THIS^.testisEqualToIgnoreCase(
	stringToTest := 'UPPERCASE',
	expectedString := 'UPPERCASE'
);
THIS^.testisEqualToIgnoreCase(
	stringToTest := 'lowercase',
	expectedString := 'lowercase'
);
THIS^.testisEqualToIgnoreCase(
	stringToTest := 'UPPERCASE',
	expectedString := 'lowercase'
);
THIS^.testisEqualToIgnoreCase(
	stringToTest := 'lowercase',
	expectedString := 'UPPERCASE'
);
THIS^.testisEqualToIgnoreCase(
	stringToTest := 'lowercase$80$B9$C6$D4',
	expectedString := 'CASE$80$B9$C6$D4'
);

TcUnit.TEST_FINISHED();
END_METHOD

(*
short summary
==================
This test method tests ``assert.string.windows125x.IsNotEmpty``
method of CNM_AssertionInterfaces library with various inputs

.. <legal notes>

legal notes
=================
| SPDX-FileCopyrightText: © 2022 ekvip automation GmbH <info@ekvip.de>
| SPDX-License-Identifier: Apache-2.0
| For details check: Apache-2.0_

.. _Apache-2.0: https://www.apache.org/licenses/LICENSE-2.0

.. </legal notes>

*)

METHOD runIsNotEmpty : BOOL
VAR_INPUT
END_VAR
RETURN (NOT TcUnit.TEST_ORDERED(THIS^.getTestNameFor('IsNotEmpty')));

THIS^.testIsNotEmpty(
	stringToTest := ''
);
THIS^.testIsNotEmpty(
	stringToTest := 'not empty'
);
THIS^.testIsNotEmpty(
	stringToTest := '{|}~'
);
THIS^.testIsNotEmpty(
	stringToTest := '3649213469328'
);
THIS^.testIsNotEmpty(
	stringToTest := '1one!'
);
THIS^.testIsNotEmpty(
	stringToTest := '$40$n$t$$$"$''
);
THIS^.testIsNotEmpty(
	stringToTest := '$n$t'
);
THIS^.testIsEmpty(
	stringToTest := '$80$8C$A9$B9$C6$D4$F4$7E',
);
THIS^.testIsNotEmpty(
	stringToTest := 'frontmiddleback'
);
THIS^.testIsNotEmpty(
	stringToTest := 'backfrontmiddle'
);
THIS^.testIsNotEmpty(
	stringToTest := 'J;%_iTxQSk?6GfWewt}yMKh1)VXqPA@P1YQ:{EAg:8VJ,/FM;j)xJ[[AvYp/}}SzEgtfYS,1K0.5VtA+VJrB(p#55h2z##mw#F)Y@P6Jz9G@6vb=x#E!cYk(Svr@S*KiPJr1VZ6AjrNback4G=vBJd.E:=,k3!wmuGDe#ZKMD#Vx%?M_0&L0#vT]J,+)ZvU{w%8X0=:XzthmT0VG0QrwpXXCWpFxu6[b!c.BunYYfLQi.,?ut?-{jrC1phTHL)y'
);

TcUnit.TEST_FINISHED();
END_METHOD

(*
short summary
==================
This test method tests ``assert.string.windows125x.isNotEqualTo``
method of CNM_AssertionInterfaces library with various inputs

.. <legal notes>

legal notes
=================
| SPDX-FileCopyrightText: © 2022 ekvip automation GmbH <info@ekvip.de>
| SPDX-License-Identifier: Apache-2.0
| For details check: Apache-2.0_

.. _Apache-2.0: https://www.apache.org/licenses/LICENSE-2.0

.. </legal notes>

*)


METHOD runIsNotEqualTo : BOOL
VAR_INPUT
END_VAR
RETURN (NOT TcUnit.TEST_ORDERED(THIS^.getTestNameFor('isNotEqualTo')));

THIS^.testisNotEqualTo(
	stringToTest := '',
	expectedString := ''
);
THIS^.testisNotEqualTo(
	stringToTest := 'not empty',
	expectedString := ''
);
THIS^.testisNotEqualTo(
	stringToTest := '',
	expectedString := 'not empty'
);
THIS^.testisNotEqualTo(
	stringToTest := 'not empty',
	expectedString := 'not'
);
THIS^.testisNotEqualTo(
	stringToTest := 'not empty',
	expectedString := 'not empty'
);
THIS^.testisNotEqualTo(
	stringToTest := '{|}~',
	expectedString := '3649213469328'
);
THIS^.testisNotEqualTo(
	stringToTest := '1one!',
	expectedString := '1one'
);
THIS^.testisNotEqualTo(
	stringToTest := '1one!',
	expectedString := '1one!'
);

THIS^.testisNotEqualTo(
	stringToTest := '$40$n$t$$$"$'',
	expectedString := '$n$t'
);
THIS^.testisNotEqualTo(
	stringToTest := '$40$n$t$$$"$'',
	expectedString := '$40$n$t$$$"$''
);
THIS^.testIsNotEqualTo(
	stringToTest := '$80$8C$A9$B9$C6$D4$F4$7E',
	expectedString := '$B9$C6$D4'
);
THIS^.testIsNotEqualTo(
	stringToTest := '$80$8C$A9$B9$C6$D4$F4$7E',
	expectedString := '$80$B9$C6$D4'
);
THIS^.testisNotEqualTo(
	stringToTest := 'frontmiddleback',
	expectedString := 'back'
);
THIS^.testisNotEqualTo(
	stringToTest := 'frontmiddleback',
	expectedString := 'frontmiddlebackfront'
);
THIS^.testisNotEqualTo(
	stringToTest := 'backfrontmiddle',
	expectedString := 'backmiddle'
);
THIS^.testisNotEqualTo(
	stringToTest := 'J;%_iTxQSk?6GfWewt}yMKh1)VXqPA@P1YQ:{EAg:8VJ,/FM;j)xJ[[AvYp/}}SzEgtfYS,1K0.5VtA+VJrB(p#55h2z##mw#F)Y@P6Jz9G@6vb=x#E!cYk(Svr@S*KiPJr1VZ6AjrNback4G=vBJd.E:=,k3!wmuGDe#ZKMD#Vx%?M_0&L0#vT]J,+)ZvU{w%8X0=:XzthmT0VG0QrwpXXCWpFxu6[b!c.BunYYfLQi.,?ut?-{jrC1phTHL)y',
	expectedString := 'J;%_iTxQSk?6GfWewt}yMKh1)VXqPA@P1YQ:{EAg:8VJ,/FM;j)xJ[[AvYp/}}SzEgtfYS,1K0.5VtA+VJrB(p#55h2z##mw#F)Y@P6Jz9G@6vb=x#E!cYk(Svr@S*KiPJr1VZ6AjrNback4G=vBJd.E:=,k3!wmuGDe#ZKMD#Vx%?M_0&L0#vT]J,+)ZvU{w%8X0=:XzthmT0VG0QrwpXXCWpFxu6[b!c.BunYYfLQi.,?ut?-{jrC1phTHL)y'
);
THIS^.testisNotEqualTo(
	stringToTest := 'J;%_iTxQSk?6GfWewt}yMKh1)VXqPA@P1YQ:{EAg:8VJ,/FM;j)xJ[[AvYp/}}SzEgtfYS,1K0.5VtA+VJrB(p#55h2z##mw#F)Y@P6Jz9G@6vb=x#E!cYk(Svr@S*KiPJr1VZ6AjrNback4G=vBJd.E:=,k3!wmuGDe#ZKMD#Vx%?M_0&L0#vT]J,+)ZvU{w%8X0=:XzthmT0VG0QrwpXXCWpFxu6[b!c.BunYYfLQi.,?ut?-{jrC1phTHL)y',
	expectedString := 'J;%_iTxQSk?6GfWewt}yMKh1)VXqPA@P1YQ:{EAg:8VJ,/FM;j)xJ[[AvYp/}}SzEgtfYS,1K0.5VtA+VJrB(p#55h2z##mw#F)Y@P6Jz9G@6vb=x#E!cYk(Svr@S*KiPJr1VZ6AjrNback4G=vBJd.E:=,k3!wmuGDe#ZKMD#Vx%?M_0&L0#vT]J,+)ZvU{w%8X0=:XzthmT0VG0QrwpXXCWpFxu6[b!c.BunYYfLQi.,?ut?-{jrC1phTHL)x'
);

THIS^.testisNotEqualToIgnoreCase(
	stringToTest := 'UPPERCASE',
	expectedString := 'UPPERCASE'
);
THIS^.testisNotEqualToIgnoreCase(
	stringToTest := 'lowercase',
	expectedString := 'lowercase'
);
THIS^.testisNotEqualToIgnoreCase(
	stringToTest := 'UPPERCASE',
	expectedString := 'lowercase'
);
THIS^.testisNotEqualToIgnoreCase(
	stringToTest := 'lowercase',
	expectedString := 'UPPERCASE'
);
THIS^.testisNotEqualToIgnoreCase(
	stringToTest := 'lowercase$80$B9$C6$D4',
	expectedString := 'CASE$80$B9$C6$D4'
);

TcUnit.TEST_FINISHED();
END_METHOD

(*
short summary
==================
This test method tests ``assert.string.windows125x.lengthIsBetween``
method of CNM_AssertionInterfaces library with various inputs

.. <legal notes>

legal notes
=================
| SPDX-FileCopyrightText: © 2022 ekvip automation GmbH <info@ekvip.de>
| SPDX-License-Identifier: Apache-2.0
| For details check: Apache-2.0_

.. _Apache-2.0: https://www.apache.org/licenses/LICENSE-2.0

.. </legal notes>

*)


METHOD runLengthIsBetween : BOOL
VAR_INPUT
END_VAR
RETURN (NOT TcUnit.TEST_ORDERED(THIS^.getTestNameFor('lengthIsBetween')));

THIS^.testLengthIsBetween(
	stringToTest := '',
	maxLength := 3,
	minLength := 0
);
THIS^.testLengthIsBetween(
	stringToTest := '',
	maxLength := 3,
	minLength := 1
);
THIS^.testLengthIsBetween(
	stringToTest := 'not empty',
	maxLength := 9,
	minLength := 0
);
THIS^.testLengthIsBetween(
	stringToTest := 'not empty',
	maxLength := 3,
	minLength := 3
);
THIS^.testLengthIsBetween(
	stringToTest := '{|}~',
	maxLength := 3,
	minLength := 3
);
THIS^.testLengthIsBetween(
	stringToTest := '{|}~',
	maxLength := 3,
	minLength := 4
);
THIS^.testLengthIsBetween(
	stringToTest := '1one!',
	maxLength := 5,
	minLength := 4
);
THIS^.testLengthIsBetween(
	stringToTest := '1one!',
	maxLength := 4,
	minLength := 3
);
THIS^.testLengthIsBetween(
	stringToTest := '$40$n$t$$$"$'',
	maxLength := 6,
	minLength := 3
);
THIS^.testLengthIsBetween(
	stringToTest := '$40$n$t$$$"$'',
	maxLength := 10,
	minLength := 7
);
THIS^.testLengthIsBetween(
	stringToTest := '$80$8C$A9$B9$C6$D4$F4$7E',
	maxLength := 8,
	minLength := 7
);
THIS^.testLengthIsBetween(
	stringToTest := '$80$8C$A9$B9$C6$D4$F4$7E',
	maxLength := 9,
	minLength := 7
);
THIS^.testLengthIsBetween(
	stringToTest := '$80$8C$A9$B9$C6$D4$F4$7E',
	maxLength := 10,
	minLength := 9
);
THIS^.testLengthIsBetween(
	stringToTest := '$80$8C$A9$B9$C6$D4$F4$7E',
	maxLength := 8,
	minLength := 9
);
THIS^.testLengthIsBetween(
	stringToTest := 'J;%_iTxQSk?6GfWewt}yMKh1)VXqPA@P1YQ:{EAg:8VJ,/FM;j)xJ[[AvYp/}}SzEgtfYS,1K0.5VtA+VJrB(p#55h2z##mw#F)Y@P6Jz9G@6vb=x#E!cYk(Svr@S*KiPJr1VZ6AjrNback4G=vBJd.E:=,k3!wmuGDe#ZKMD#Vx%?M_0&L0#vT]J,+)ZvU{w%8X0=:XzthmT0VG0QrwpXXCWpFxu6[b!c.BunYYfLQi.,?ut?-{jrC1phTHL)y',
	maxLength := 255,
	minLength := 7
);
THIS^.testLengthIsBetween(
	stringToTest := 'J;%_iTxQSk?6GfWewt}yMKh1)VXqPA@P1YQ:{EAg:8VJ,/FM;j)xJ[[AvYp/}}SzEgtfYS,1K0.5VtA+VJrB(p#55h2z##mw#F)Y@P6Jz9G@6vb=x#E!cYk(Svr@S*KiPJr1VZ6AjrNback4G=vBJd.E:=,k3!wmuGDe#ZKMD#Vx%?M_0&L0#vT]J,+)ZvU{w%8X0=:XzthmT0VG0QrwpXXCWpFxu6[b!c.BunYYfLQi.,?ut?-{jrC1phTHL)y',
	maxLength := 254,
	minLength := 7
);
THIS^.testLengthIsBetween(
	stringToTest := 'J;%_iTxQSk?6GfWewt}yMKh1)VXqPA@P1YQ:{EAg:8VJ,/FM;j)xJ[[AvYp/}}SzEgtfYS,1K0.5VtA+VJrB(p#55h2z##mw#F)Y@P6Jz9G@6vb=x#E!cYk(Svr@S*KiPJr1VZ6AjrNback4G=vBJd.E:=,k3!wmuGDe#ZKMD#Vx%?M_0&L0#vT]J,+)ZvU{w%8X0=:XzthmT0VG0QrwpXXCWpFxu6[b!c.BunYYfLQi.,?ut?-{jrC1phTHL)y',
	maxLength := 255,
	minLength := 255
);

TcUnit.TEST_FINISHED();
END_METHOD

(*
short summary
==================
This test method tests ``assert.string.windows125x.lengthIsExact``
method of CNM_AssertionInterfaces library with various inputs

.. <legal notes>

legal notes
=================
| SPDX-FileCopyrightText: © 2022 ekvip automation GmbH <info@ekvip.de>
| SPDX-License-Identifier: Apache-2.0
| For details check: Apache-2.0_

.. _Apache-2.0: https://www.apache.org/licenses/LICENSE-2.0

.. </legal notes>

*)


METHOD runLengthIsExact : BOOL
VAR_INPUT
END_VAR
RETURN (NOT TcUnit.TEST_ORDERED(THIS^.getTestNameFor('lengthIsExact')));

THIS^.testLengthIsExact(
	stringToTest := '',
	expectedLength := 0
);
THIS^.testLengthIsExact(
	stringToTest := '',
	expectedLength := 1
);
THIS^.testLengthIsExact(
	stringToTest := 'not empty',
	expectedLength := 9
);
THIS^.testLengthIsExact(
	stringToTest := 'not empty',
	expectedLength := 8
);
THIS^.testLengthIsExact(
	stringToTest := 'not empty',
	expectedLength := 10
);
THIS^.testLengthIsExact(
	stringToTest := '{|}~',
	expectedLength := 4
);
THIS^.testLengthIsExact(
	stringToTest := '{|}~',
	expectedLength := 40
);
THIS^.testLengthIsExact(
	stringToTest := '1one!',
	expectedLength := 5
);
THIS^.testLengthIsExact(
	stringToTest := '1one!',
	expectedLength := 6
);
THIS^.testLengthIsExact(
	stringToTest := '$40$n$t$$$"$'',
	expectedLength := 6
);
THIS^.testLengthIsExact(
	stringToTest := '$40$n$t$$$"$'',
	expectedLength := 7
);
THIS^.testLengthIsExact(
	stringToTest := '$80$8C$A9$B9$C6$D4$F4$7E',
	expectedLength := 8
);
THIS^.testLengthIsExact(
	stringToTest := '$80$8C$A9$B9$C6$D4$F4$7E',
	expectedLength := 9
);
THIS^.testLengthIsExact(
	stringToTest := '$80$8C$A9$B9$C6$D4$F4$7E',
	expectedLength := 7
);
THIS^.testLengthIsExact(
	stringToTest := 'J;%_iTxQSk?6GfWewt}yMKh1)VXqPA@P1YQ:{EAg:8VJ,/FM;j)xJ[[AvYp/}}SzEgtfYS,1K0.5VtA+VJrB(p#55h2z##mw#F)Y@P6Jz9G@6vb=x#E!cYk(Svr@S*KiPJr1VZ6AjrNback4G=vBJd.E:=,k3!wmuGDe#ZKMD#Vx%?M_0&L0#vT]J,+)ZvU{w%8X0=:XzthmT0VG0QrwpXXCWpFxu6[b!c.BunYYfLQi.,?ut?-{jrC1phTHL)y',
	expectedLength := 255
);
THIS^.testLengthIsExact(
	stringToTest := 'J;%_iTxQSk?6GfWewt}yMKh1)VXqPA@P1YQ:{EAg:8VJ,/FM;j)xJ[[AvYp/}}SzEgtfYS,1K0.5VtA+VJrB(p#55h2z##mw#F)Y@P6Jz9G@6vb=x#E!cYk(Svr@S*KiPJr1VZ6AjrNback4G=vBJd.E:=,k3!wmuGDe#ZKMD#Vx%?M_0&L0#vT]J,+)ZvU{w%8X0=:XzthmT0VG0QrwpXXCWpFxu6[b!c.BunYYfLQi.,?ut?-{jrC1phTHL)y',
	expectedLength := 254
);

TcUnit.TEST_FINISHED();
END_METHOD

(*
short summary
==================
This test method tests ``assert.string.windows125x.lengthIsMax``
method of CNM_AssertionInterfaces library with various inputs

.. <legal notes>

legal notes
=================
| SPDX-FileCopyrightText: © 2022 ekvip automation GmbH <info@ekvip.de>
| SPDX-License-Identifier: Apache-2.0
| For details check: Apache-2.0_

.. _Apache-2.0: https://www.apache.org/licenses/LICENSE-2.0

.. </legal notes>

*)


METHOD runLengthIsMax : BOOL
VAR_INPUT
END_VAR
RETURN (NOT TcUnit.TEST_ORDERED(THIS^.getTestNameFor('lengthIsMax')));

THIS^.testLengthIsMax(
	stringToTest := '',
	expectedLength := 0
);
THIS^.testLengthIsMax(
	stringToTest := '',
	expectedLength := 1
);
THIS^.testLengthIsMax(
	stringToTest := 'not empty',
	expectedLength := 9
);
THIS^.testLengthIsMax(
	stringToTest := 'not empty',
	expectedLength := 8
);
THIS^.testLengthIsMax(
	stringToTest := 'not empty',
	expectedLength := 10
);
THIS^.testLengthIsMax(
	stringToTest := '{|}~',
	expectedLength := 4
);
THIS^.testLengthIsMax(
	stringToTest := '{|}~',
	expectedLength := 40
);
THIS^.testLengthIsMax(
	stringToTest := '{|}~',
	expectedLength := 3
);
THIS^.testLengthIsMax(
	stringToTest := '1one!',
	expectedLength := 5
);
THIS^.testLengthIsMax(
	stringToTest := '1one!',
	expectedLength := 4
);
THIS^.testLengthIsMax(
	stringToTest := '$40$n$t$$$"$'',
	expectedLength := 6
);
THIS^.testLengthIsMax(
	stringToTest := '$40$n$t$$$"$'',
	expectedLength := 5
);
THIS^.testLengthIsMax(
	stringToTest := '$80$8C$A9$B9$C6$D4$F4$7E',
	expectedLength := 8
);
THIS^.testLengthIsMax(
	stringToTest := '$80$8C$A9$B9$C6$D4$F4$7E',
	expectedLength := 9
);
THIS^.testLengthIsMax(
	stringToTest := '$80$8C$A9$B9$C6$D4$F4$7E',
	expectedLength := 7
);
THIS^.testLengthIsMax(
	stringToTest := 'J;%_iTxQSk?6GfWewt}yMKh1)VXqPA@P1YQ:{EAg:8VJ,/FM;j)xJ[[AvYp/}}SzEgtfYS,1K0.5VtA+VJrB(p#55h2z##mw#F)Y@P6Jz9G@6vb=x#E!cYk(Svr@S*KiPJr1VZ6AjrNback4G=vBJd.E:=,k3!wmuGDe#ZKMD#Vx%?M_0&L0#vT]J,+)ZvU{w%8X0=:XzthmT0VG0QrwpXXCWpFxu6[b!c.BunYYfLQi.,?ut?-{jrC1phTHL)y',
	expectedLength := 255
);
THIS^.testLengthIsMax(
	stringToTest := 'J;%_iTxQSk?6GfWewt}yMKh1)VXqPA@P1YQ:{EAg:8VJ,/FM;j)xJ[[AvYp/}}SzEgtfYS,1K0.5VtA+VJrB(p#55h2z##mw#F)Y@P6Jz9G@6vb=x#E!cYk(Svr@S*KiPJr1VZ6AjrNback4G=vBJd.E:=,k3!wmuGDe#ZKMD#Vx%?M_0&L0#vT]J,+)ZvU{w%8X0=:XzthmT0VG0QrwpXXCWpFxu6[b!c.BunYYfLQi.,?ut?-{jrC1phTHL)y',
	expectedLength := 254
);

TcUnit.TEST_FINISHED();
END_METHOD

(*
short summary
==================
This test method tests ``assert.string.windows125x.lengthIsMin``
method of CNM_AssertionInterfaces library with various inputs

.. <legal notes>

legal notes
=================
| SPDX-FileCopyrightText: © 2022 ekvip automation GmbH <info@ekvip.de>
| SPDX-License-Identifier: Apache-2.0
| For details check: Apache-2.0_

.. _Apache-2.0: https://www.apache.org/licenses/LICENSE-2.0

.. </legal notes>

*)


METHOD runLengthIsMin : BOOL
VAR_INPUT
END_VAR
RETURN (NOT TcUnit.TEST_ORDERED(THIS^.getTestNameFor('lengthIsMin')));

THIS^.testLengthIsMin(
	stringToTest := '',
	expectedLength := 0
);
THIS^.testLengthIsMin(
	stringToTest := '',
	expectedLength := 1
);
THIS^.testLengthIsMin(
	stringToTest := 'not empty',
	expectedLength := 9
);
THIS^.testLengthIsMin(
	stringToTest := 'not empty',
	expectedLength := 8
);
THIS^.testLengthIsMin(
	stringToTest := 'not empty',
	expectedLength := 10
);
THIS^.testLengthIsMin(
	stringToTest := '{|}~',
	expectedLength := 4
);
THIS^.testLengthIsMin(
	stringToTest := '{|}~',
	expectedLength := 40
);
THIS^.testLengthIsMin(
	stringToTest := '{|}~',
	expectedLength := 3
);
THIS^.testLengthIsMin(
	stringToTest := '1one!',
	expectedLength := 5
);
THIS^.testLengthIsMin(
	stringToTest := '1one!',
	expectedLength := 6
);
THIS^.testLengthIsMin(
	stringToTest := '$40$n$t$$$"$'',
	expectedLength := 6
);
THIS^.testLengthIsMin(
	stringToTest := '$40$n$t$$$"$'',
	expectedLength := 7
);
THIS^.testLengthIsMin(
	stringToTest := '$80$8C$A9$B9$C6$D4$F4$7E',
	expectedLength := 8
);
THIS^.testLengthIsMin(
	stringToTest := '$80$8C$A9$B9$C6$D4$F4$7E',
	expectedLength := 9
);
THIS^.testLengthIsMin(
	stringToTest := '$80$8C$A9$B9$C6$D4$F4$7E',
	expectedLength := 7
);
THIS^.testLengthIsMin(
	stringToTest := 'J;%_iTxQSk?6GfWewt}yMKh1)VXqPA@P1YQ:{EAg:8VJ,/FM;j)xJ[[AvYp/}}SzEgtfYS,1K0.5VtA+VJrB(p#55h2z##mw#F)Y@P6Jz9G@6vb=x#E!cYk(Svr@S*KiPJr1VZ6AjrNback4G=vBJd.E:=,k3!wmuGDe#ZKMD#Vx%?M_0&L0#vT]J,+)ZvU{w%8X0=:XzthmT0VG0QrwpXXCWpFxu6[b!c.BunYYfLQi.,?ut?-{jrC1phTHL)y',
	expectedLength := 255
);
THIS^.testLengthIsMin(
	stringToTest := 'J;%_iTxQSk?6GfWewt}yMKh1)VXqPA@P1YQ:{EAg:8VJ,/FM;j)xJ[[AvYp/}}SzEgtfYS,1K0.5VtA+VJrB(p#55h2z##mw#F)Y@P6Jz9G@6vb=x#E!cYk(Svr@S*KiPJr1VZ6AjrNback4G=vBJd.E:=,k3!wmuGDe#ZKMD#Vx%?M_0&L0#vT]J,+)ZvU{w%8X0=:XzthmT0VG0QrwpXXCWpFxu6[b!c.BunYYfLQi.,?ut?-{jrC1phTHL)y',
	expectedLength := 254
);

TcUnit.TEST_FINISHED();
END_METHOD

(*
short summary
==================
This test method tests ``assert.string.windows125x.startsWith``
method of CNM_AssertionInterfaces library with various inputs

.. <legal notes>

legal notes
=================
| SPDX-FileCopyrightText: © 2022 ekvip automation GmbH <info@ekvip.de>
| SPDX-License-Identifier: Apache-2.0
| For details check: Apache-2.0_

.. _Apache-2.0: https://www.apache.org/licenses/LICENSE-2.0

.. </legal notes>

*)


METHOD runStartsWith : BOOL
VAR_INPUT
END_VAR
RETURN (NOT TcUnit.TEST_ORDERED(THIS^.getTestNameFor('startsWith')));

THIS^.testStartsWith(
	stringToTest := '',
	expectedString := ''
);
THIS^.testStartsWith(
	stringToTest := 'not empty',
	expectedString := ''
);
THIS^.testStartsWith(
	stringToTest := '',
	expectedString := 'not empty'
);
THIS^.testStartsWith(
	stringToTest := 'not empty',
	expectedString := 'not empty'
);
THIS^.testStartsWith(
	stringToTest := '{|}~',
	expectedString := '3649213469328'
);
THIS^.testStartsWith(
	stringToTest := '1one!',
	expectedString := '1'
);
THIS^.testStartsWith(
	stringToTest := '1one!',
	expectedString := 'one'
);
THIS^.testStartsWith(
	stringToTest := '1one!',
	expectedString := '!'
);
THIS^.testStartsWith(
	stringToTest := '$40$n$t$$$"$'',
	expectedString := '$n$t'
);
THIS^.testStartsWith(
	stringToTest := '$n$t$40$$$"$'',
	expectedString := '$n$t'
);
THIS^.testStartsWith(
	stringToTest := '$80$8C$A9$B9$C6$D4$F4$7E',
	expectedString := '$B9$C6$D4'
);
THIS^.testStartsWith(
	stringToTest := '$80$8C$A9$B9$C6$D4$F4$7E',
	expectedString := '$80$8C$A9$B9'
);
THIS^.testStartsWith(
	stringToTest := 'frontmiddleback',
	expectedString := 'front'
);
THIS^.testStartsWith(
	stringToTest := 'frontmiddleback',
	expectedString := 'frontmiddlebackfront'
);
THIS^.testStartsWith(
	stringToTest := 'backfrontmiddle',
	expectedString := 'backmiddle'
);
THIS^.testStartsWith(
	stringToTest := 'J;%_iTxQSk?6GfWewt}yMKh1)VXqPA@P1YQ:{EAg:8VJ,/FM;j)xJ[[AvYp/}}SzEgtfYS,1K0.5VtA+VJrB(p#55h2z##mw#F)Y@P6Jz9G@6vb=x#E!cYk(Svr@S*KiPJr1VZ6AjrNback4G=vBJd.E:=,k3!wmuGDe#ZKMD#Vx%?M_0&L0#vT]J,+)ZvU{w%8X0=:XzthmT0VG0QrwpXXCWpFxu6[b!c.BunYYfLQi.,?ut?-{jrC1phTHL)y',
	expectedString := 'J;%_iTxQSk?6GfWewt}yMKh1)VXqPA@P1YQ:{EAg:8VJ,/FM;j)xJ[[AvYp/}}SzEgtfYS,1K0.5VtA+VJrB(p#55h2z##mw#F)Y@P6Jz9G@6vb=x#E!cYk(Svr@S*KiPJr1VZ6AjrNback4G=vBJd.E:=,k3!wmuGDe#ZKMD#Vx%?M_0&L0#vT]J,+)ZvU{w%8X0=:XzthmT0VG0QrwpXXCWpFxu6[b!c.BunYYfLQi.,?ut?-{jrC1phTHL)y'
);
THIS^.testStartsWith(
	stringToTest := 'J;%_iTxQSk?6GfWewt}yMKh1)VXqPA@P1YQ:{EAg:8VJ,/FM;j)xJ[[AvYp/}}SzEgtfYS,1K0.5VtA+VJrB(p#55h2z##mw#F)Y@P6Jz9G@6vb=x#E!cYk(Svr@S*KiPJr1VZ6AjrNback4G=vBJd.E:=,k3!wmuGDe#ZKMD#Vx%?M_0&L0#vT]J,+)ZvU{w%8X0=:XzthmT0VG0QrwpXXCWpFxu6[b!c.BunYYfLQi.,?ut?-{jrC1phTHL)y',
	expectedString := 'J;%_iTxQSk?6GfWewt}yMKh1)VXqPA@P1YQ:{EAg:8VJ,/FM;j)xJ[[AvYp/}}SzEgtfYS,1K0.5VtA+VJrB(p#55h2z##mw#F)Y@P6Jz9G@6vb=x#E!cYk(Svr@S*KiPJr1VZ6AjrNback4G=vBJd.E:=,k3!wmuGDe#ZKMD#Vx%?M_0&L0#vT]J,+)ZvU{w%8X0=:XzthmT0VG0QrwpXXCWpFxu6[b!c.BunYYfLQi.,?ut?-{jrC1phTHL)x'
);

THIS^.testStartsWithIgnoreCase(
	stringToTest := 'UPPERCASE',
	expectedString := 'UPPER'
);
THIS^.testStartsWithIgnoreCase(
	stringToTest := 'lowercase',
	expectedString := 'lower'
);
THIS^.testStartsWithIgnoreCase(
	stringToTest := 'UPPERCASE',
	expectedString := 'upper'
);
THIS^.testStartsWithIgnoreCase(
	stringToTest := 'lowercase',
	expectedString := 'LOWER'
);
THIS^.testStartsWithIgnoreCase(
	stringToTest := 'lower',
	expectedString := 'UPPER'
);
THIS^.testStartsWithIgnoreCase(
	stringToTest := '$80$B9$C6$D4lowercase',
	expectedString := '$80$B9$C6$D4LOWER'
);

THIS^.testStartsWithTrim(
	stringToTest := '$tfrontmiddleback',
	expectedString := 'front',
	expectedAssertionResult := TRUE
);
THIS^.testStartsWithTrim(
	stringToTest := 'frontmiddleback',
	expectedString := '$tfront',
	expectedAssertionResult := TRUE
);
THIS^.testStartsWithTrim(
	stringToTest := '$20frontmiddleback',
	expectedString := 'front',
	expectedAssertionResult := TRUE
);
THIS^.testStartsWithTrim(
	stringToTest := 'frontmiddleback',
	expectedString := '$20front',
	expectedAssertionResult := TRUE
);
THIS^.testStartsWithTrim(
	stringToTest := '$t$n$r$p$lfrontmiddleback',
	expectedString := 'front$25',
	expectedAssertionResult := FALSE
);
THIS^.testStartsWithTrim(
	stringToTest := '$t$n$r$p$lfrontmiddleback',
	expectedString := 'front',
	expectedAssertionResult := TRUE
);
THIS^.testStartsWithTrim(
	stringToTest := '$20$80$B9$C6$D4frontmiddleback',
	expectedString := '$80$B9$C6$D4front',
	expectedAssertionResult := TRUE
);
THIS^.testStartsWithTrim(
	stringToTest := '$20$80$B9$B9$C6$D4frontmiddleback',
	expectedString := '$80$B9$C6$D4front',
	expectedAssertionResult := FALSE
);

TcUnit.TEST_FINISHED();
END_METHOD

(*
short summary
==================
This test method tests ``assert.string.windows125x.contains``
method of CNM_AssertionInterfaces library with various inputs

.. <legal notes>

legal notes
=================
| SPDX-FileCopyrightText: © 2022 ekvip automation GmbH <info@ekvip.de>
| SPDX-License-Identifier: Apache-2.0
| For details check: Apache-2.0_

.. _Apache-2.0: https://www.apache.org/licenses/LICENSE-2.0

.. </legal notes>

*)


METHOD testContains : BOOL
VAR_INPUT
	(* for the test it's the parameter ``stringToCheck`` *)
	stringToTest 	:Tc2_System.T_MaxString;
	(* for the test it's the parameter ``searchString`` *)
	expectedString 	:Tc2_System.T_MaxString;
END_VAR
VAR 
	(* just the expectation if the assertion to test must be worng or true *)
	assertionIsWrong		:BOOL;
	(* contains the format string for the test message *)
	message					:Tc2_System.T_MaxString;
	(* used for placeholder string if stringToTest can't be printed *)
	stringToTestAsString 	:Tc2_System.T_MaxString := stringToTest;
	(* used for placeholder string if expectedString can't be printed *)
	expectedStringAsString 	:Tc2_System.T_MaxString := expectedString;
	(* TwinCAT printf with the test message *)
	messageStringBuilder	:Tc2_Utilities.FB_FormatString;
END_VAR
THIS^.assertorContainer.resetAssertor();

assertionIsWrong := ((
		Tc2_Standard.FIND(
			stringToTest,
			expectedString
		) = 0
	) AND (
		Tc2_Standard.LEN(
			expectedString
		) <> 0
	)
);

message := SEL(
	assertionIsWrong,
	'stringToCheck is $'%s$' searchString is $'%s$' assertion must be TRUE', 
	'stringToCheck is $'%s$' searchString is $'%s$' assertion must be FALSE'
);

IF (
		Tc2_Standard.LEN(stringToTest) = TO_DINT(Tc2_System.MAX_STRING_LENGTH)
) THEN
	stringToTestAsString := 'String with Tc2_System.MAX_STRING_LENGTH characters';
END_IF
IF (
		Tc2_Standard.LEN(expectedString) = TO_DINT(Tc2_System.MAX_STRING_LENGTH)
) THEN
	expectedStringAsString := 'String with Tc2_System.MAX_STRING_LENGTH characters';
END_IF

messageStringBuilder(
	sFormat := message,
	arg1 := THIS^.AnyToArg(stringToTestAsString),
	arg2 := THIS^.AnyToArg(expectedStringAsString)
);


THIS^.assertorContainer.assertor.assert.strings.windows125x.contains(
	stringToCheck := stringToTest,
	searchString := expectedString,
	ignoreCases := FALSE,
	message			:= ''
);
   
THIS^.AssertEquals_BOOL(
	Expected 	:= assertionIsWrong,
	Actual 		:= THIS^.assertorContainer.wasAssertionWrong,
	Message 	:= messageStringBuilder.sOut
);

THIS^.assertorContainer.assertor.assert.strings.windows125x.contains(
	stringToCheck := stringToTest,
	searchString := expectedString,
	ignoreCases := FALSE,
	sbcsType := Tc2_Utilities.E_SBCSType.eSBCS_CentralEuropean,
	message			:= ''
);

THIS^.AssertEquals_BOOL(
	Expected 	:= assertionIsWrong,
	Actual 		:= THIS^.assertorContainer.wasAssertionWrong,
	Message 	:= messageStringBuilder.sOut
);
END_METHOD

(*
short summary
==================
This test method tests ``assert.string.windows125x.contains``
method of CNM_AssertionInterfaces library with various inputs

.. <legal notes>

legal notes
=================
| SPDX-FileCopyrightText: © 2022 ekvip automation GmbH <info@ekvip.de>
| SPDX-License-Identifier: Apache-2.0
| For details check: Apache-2.0_

.. _Apache-2.0: https://www.apache.org/licenses/LICENSE-2.0

.. </legal notes>

*)


METHOD testContainsIgnoreCase : BOOL
VAR_INPUT
	(* for the test it's the parameter ``stringToCheck`` *)
	stringToTest 	:Tc2_System.T_MaxString;
	(* for the test it's the parameter ``searchString`` *)
	expectedString 	:Tc2_System.T_MaxString;
END_VAR
VAR 
	(* just the expectation if the assertion to test must be worng or true *)
	assertionIsWrong		:BOOL;
	(* contains the format string for the test message *)
	message					:Tc2_System.T_MaxString;
	(* contains ´´stringToTest´´ in upper case *)
	upperStringToTest		:Tc2_System.T_MaxString := stringToTest;
	(* contains ´´expectedString´´ in upper case *)
	upperExpectedString		:Tc2_System.T_MaxString := expectedString;
	(* used for placeholder string if stringToTest can't be printed *)
	stringToTestAsString 	:Tc2_System.T_MaxString := stringToTest;
	(* used for placeholder string if expectedString can't be printed *)
	expectedStringAsString 	:Tc2_System.T_MaxString := expectedString;
	(* TwinCAT printf with the test message *)
	messageStringBuilder	:Tc2_Utilities.FB_FormatString;
END_VAR
THIS^.assertorContainer.resetAssertor();

// both Strings to upper case
upperStringToTest := Tc2_Utilities.F_ToUCase(upperStringToTest);
upperExpectedString := Tc2_Utilities.F_ToUCase(upperExpectedString);

assertionIsWrong := ((
		Tc2_Standard.FIND(
			upperStringToTest,
			upperExpectedString
		) = 0
	) AND (
		Tc2_Standard.LEN(
			upperExpectedString
		) <> 0
	)
);

message := SEL(
	assertionIsWrong,
	'stringToCheck is $'%s$' searchString is $'%s$' assertion must be TRUE', 
	'stringToCheck is $'%s$' searchString is $'%s$' assertion must be FALSE'
);

IF (
		Tc2_Standard.LEN(stringToTest) = TO_DINT(Tc2_System.MAX_STRING_LENGTH)
) THEN
	stringToTestAsString := 'String with Tc2_System.MAX_STRING_LENGTH characters';
END_IF
IF (
		Tc2_Standard.LEN(expectedString) = TO_DINT(Tc2_System.MAX_STRING_LENGTH)
) THEN
	expectedStringAsString := 'String with Tc2_System.MAX_STRING_LENGTH characters';
END_IF

messageStringBuilder(
	sFormat := message,
	arg1 := THIS^.AnyToArg(stringToTestAsString),
	arg2 := THIS^.AnyToArg(expectedStringAsString)
);


THIS^.assertorContainer.assertor.assert.strings.windows125x.contains(
	stringToCheck := stringToTest,
	searchString := expectedString,
	ignoreCases := TRUE,
	message			:= ''
);
   
THIS^.AssertEquals_BOOL(
	Expected 	:= assertionIsWrong,
	Actual 		:= THIS^.assertorContainer.wasAssertionWrong,
	Message 	:= messageStringBuilder.sOut
);

THIS^.assertorContainer.assertor.assert.strings.windows125x.contains(
	stringToCheck := stringToTest,
	searchString := expectedString,
	ignoreCases := TRUE,
	sbcsType := Tc2_Utilities.E_SBCSType.eSBCS_CentralEuropean,
	message			:= ''
);

THIS^.AssertEquals_BOOL(
	Expected 	:= assertionIsWrong,
	Actual 		:= THIS^.assertorContainer.wasAssertionWrong,
	Message 	:= messageStringBuilder.sOut
);
END_METHOD

(*
short summary
==================
This test method tests ``assert.string.windows125x.containsNo``
method of CNM_AssertionInterfaces library with various inputs

.. <legal notes>

legal notes
=================
| SPDX-FileCopyrightText: © 2022 ekvip automation GmbH <info@ekvip.de>
| SPDX-License-Identifier: Apache-2.0
| For details check: Apache-2.0_

.. _Apache-2.0: https://www.apache.org/licenses/LICENSE-2.0

.. </legal notes>

*)


METHOD testContainsNo : BOOL
VAR_INPUT
	(* for the test it's the parameter ``stringToCheck`` *)
	stringToTest 	:Tc2_System.T_MaxString;
	(* for the test it's the parameter ``searchString`` *)
	expectedString 	:Tc2_System.T_MaxString;
END_VAR
VAR 
	(* just the expectation if the assertion to test must be worng or true *)
	assertionIsWrong		:BOOL;
	(* contains the format string for the test message *)
	message					:Tc2_System.T_MaxString;
	(* used for placeholder string if stringToTest can't be printed *)
	stringToTestAsString 	:Tc2_System.T_MaxString := stringToTest;
	(* used for placeholder string if expectedString can't be printed *)
	expectedStringAsString 	:Tc2_System.T_MaxString := expectedString;
	(* TwinCAT printf with the test message *)
	messageStringBuilder	:Tc2_Utilities.FB_FormatString;
END_VAR
THIS^.assertorContainer.resetAssertor();

assertionIsWrong := ((
		Tc2_Standard.FIND(
			stringToTest,
			expectedString
		) > 0
	) OR ( Tc2_Standard.LEN( expectedString ) = 0)
);

message := SEL(
	assertionIsWrong,
	'stringToCheck is $'%s$' searchString is $'%s$' assertion must be TRUE', 
	'stringToCheck is $'%s$' searchString is $'%s$' assertion must be FALSE'
);

IF (
		Tc2_Standard.LEN(stringToTest) = TO_DINT(Tc2_System.MAX_STRING_LENGTH)
) THEN
	stringToTestAsString := 'String with Tc2_System.MAX_STRING_LENGTH characters';
END_IF
IF (
		Tc2_Standard.LEN(expectedString) = TO_DINT(Tc2_System.MAX_STRING_LENGTH)
) THEN
	expectedStringAsString := 'String with Tc2_System.MAX_STRING_LENGTH characters';
END_IF

messageStringBuilder(
	sFormat := message,
	arg1 := THIS^.AnyToArg(stringToTestAsString),
	arg2 := THIS^.AnyToArg(expectedStringAsString)
);

THIS^.assertorContainer.assertor.assert.strings.windows125x.containsNo(
	stringToCheck := stringToTest,
	searchString := expectedString,
	ignoreCases := FALSE,
	message			:= ''
);
   
THIS^.AssertEquals_BOOL(
	Expected 	:= assertionIsWrong,
	Actual 		:= THIS^.assertorContainer.wasAssertionWrong,
	Message 	:= messageStringBuilder.sOut
);

THIS^.assertorContainer.assertor.assert.strings.windows125x.containsNo(
	stringToCheck := stringToTest,
	searchString := expectedString,
	ignoreCases := FALSE,
	sbcsType := Tc2_Utilities.E_SBCSType.eSBCS_CentralEuropean,
	message			:= ''
);

THIS^.AssertEquals_BOOL(
	Expected 	:= assertionIsWrong,
	Actual 		:= THIS^.assertorContainer.wasAssertionWrong,
	Message 	:= messageStringBuilder.sOut
);
END_METHOD

(*
short summary
==================
This test method tests ``assert.string.windows125x.containsNo``
method of CNM_AssertionInterfaces library with various inputs

.. <legal notes>

legal notes
=================
| SPDX-FileCopyrightText: © 2022 ekvip automation GmbH <info@ekvip.de>
| SPDX-License-Identifier: Apache-2.0
| For details check: Apache-2.0_

.. _Apache-2.0: https://www.apache.org/licenses/LICENSE-2.0

.. </legal notes>

*)


METHOD testContainsNoIgnoreCase : BOOL
VAR_INPUT
	(* for the test it's the parameter ``stringToCheck`` *)
	stringToTest 	:Tc2_System.T_MaxString;
	(* for the test it's the parameter ``searchString`` *)
	expectedString 	:Tc2_System.T_MaxString;
END_VAR
VAR 
	(* just the expectation if the assertion to test must be worng or true *)
	assertionIsWrong		:BOOL;
	(* contains the format string for the test message *)
	message					:Tc2_System.T_MaxString;
	(* contains ´´stringToTest´´ in upper case *)
	upperStringToTest		:Tc2_System.T_MaxString := stringToTest;
	(* contains ´´expectedString´´ in upper case *)
	upperExpectedString		:Tc2_System.T_MaxString := expectedString;
	(* used for placeholder string if stringToTest can't be printed *)
	stringToTestAsString 	:Tc2_System.T_MaxString := stringToTest;
	(* used for placeholder string if expectedString can't be printed *)
	expectedStringAsString 	:Tc2_System.T_MaxString := expectedString;
	(* TwinCAT printf with the test message *)
	messageStringBuilder	:Tc2_Utilities.FB_FormatString;
END_VAR
THIS^.assertorContainer.resetAssertor();

// both Strings to upper case
upperStringToTest := Tc2_Utilities.F_ToUCase(upperStringToTest);
upperExpectedString := Tc2_Utilities.F_ToUCase(upperExpectedString);

assertionIsWrong := ((
		Tc2_Standard.FIND(
			upperStringToTest,
			upperExpectedString
		) > 0
	) OR (
		LEN(
			upperExpectedString
		) = 0
	)
);

message := SEL(
	assertionIsWrong,
	'stringToCheck is $'%s$' searchString is $'%s$' assertion must be TRUE', 
	'stringToCheck is $'%s$' searchString is $'%s$' assertion must be FALSE'
);

IF (
		Tc2_Standard.LEN(stringToTest) = TO_DINT(Tc2_System.MAX_STRING_LENGTH)
) THEN
	stringToTestAsString := 'String with Tc2_System.MAX_STRING_LENGTH characters';
END_IF
IF (
		Tc2_Standard.LEN(expectedString) = TO_DINT(Tc2_System.MAX_STRING_LENGTH)
) THEN
	expectedStringAsString := 'String with Tc2_System.MAX_STRING_LENGTH characters';
END_IF

messageStringBuilder(
	sFormat := message,
	arg1 := THIS^.AnyToArg(stringToTestAsString),
	arg2 := THIS^.AnyToArg(expectedStringAsString)
);


THIS^.assertorContainer.assertor.assert.strings.windows125x.containsNo(
	stringToCheck := stringToTest,
	searchString := expectedString,
	ignoreCases := TRUE,
	message			:= ''
);
   
THIS^.AssertEquals_BOOL(
	Expected 	:= assertionIsWrong,
	Actual 		:= THIS^.assertorContainer.wasAssertionWrong,
	Message 	:= messageStringBuilder.sOut
);

THIS^.assertorContainer.assertor.assert.strings.windows125x.containsNo(
	stringToCheck := stringToTest,
	searchString := expectedString,
	ignoreCases := TRUE,
	sbcsType := Tc2_Utilities.E_SBCSType.eSBCS_CentralEuropean,
	message			:= ''
);

THIS^.AssertEquals_BOOL(
	Expected 	:= assertionIsWrong,
	Actual 		:= THIS^.assertorContainer.wasAssertionWrong,
	Message 	:= messageStringBuilder.sOut
);
END_METHOD

(*
short summary
==================
This test method tests ``assert.string.windows125x.endsWith``
method of CNM_AssertionInterfaces library with various inputs

.. <legal notes>

legal notes
=================
| SPDX-FileCopyrightText: © 2022 ekvip automation GmbH <info@ekvip.de>
| SPDX-License-Identifier: Apache-2.0
| For details check: Apache-2.0_

.. _Apache-2.0: https://www.apache.org/licenses/LICENSE-2.0

.. </legal notes>

*)


METHOD testEndsWith : BOOL
VAR_INPUT
	(* for the test it's the parameter ``stringToCheck`` *)
	stringToTest 	:Tc2_System.T_MaxString;
	(* for the test it's the parameter ``end`` *)
	expectedString 	:Tc2_System.T_MaxString;
END_VAR
VAR 
	(* just the expectation if the assertion to test must be worng or true *)
	assertionIsWrong		:BOOL;
	(* contains the format string for the test message *)
	message					:Tc2_System.T_MaxString;
	(* used for placeholder string if stringToTest can't be printed *)
	stringToTestAsString 	:Tc2_System.T_MaxString := stringToTest;
	(* used for placeholder string if expectedString can't be printed *)
	expectedStringAsString 	:Tc2_System.T_MaxString := expectedString;
	(* TwinCAT printf with the test message *)
	messageStringBuilder	:Tc2_Utilities.FB_FormatString;
END_VAR
THIS^.assertorContainer.resetAssertor();

assertionIsWrong := ((
		Tc2_Standard.FIND(
			Tc2_Standard.RIGHT(
				stringToTest,
				Tc2_Standard.LEN(expectedString)
			),
			expectedString
		) <> 1
	) AND (
		Tc2_Standard.LEN(
				expectedString
		) <> 0
	)
);

message := SEL(
	assertionIsWrong,
	'stringToCheck is $'%s$' end is $'%s$' assertion must be TRUE', 
	'stringToCheck is $'%s$' end is $'%s$' assertion must be FALSE'
);

IF (
		Tc2_Standard.LEN(stringToTest) = TO_DINT(Tc2_System.MAX_STRING_LENGTH)
) THEN
	stringToTestAsString := 'String with Tc2_System.MAX_STRING_LENGTH characters';
END_IF
IF (
		Tc2_Standard.LEN(expectedString) = TO_DINT(Tc2_System.MAX_STRING_LENGTH)
) THEN
	expectedStringAsString := 'String with Tc2_System.MAX_STRING_LENGTH characters';
END_IF

messageStringBuilder(
	sFormat := message,
	arg1 := THIS^.AnyToArg(stringToTestAsString),
	arg2 := THIS^.AnyToArg(expectedStringAsString)
);


THIS^.assertorContainer.assertor.assert.strings.windows125x.endsWith(
	stringToCheck := stringToTest,
	end := expectedString,
	ignoreCases := FALSE,
	trim := FALSE,
	message			:= ''
);

THIS^.AssertEquals_BOOL(
	Expected 	:= assertionIsWrong,
	Actual 		:= THIS^.assertorContainer.wasAssertionWrong,
	Message 	:= messageStringBuilder.sOut
);

THIS^.assertorContainer.assertor.assert.strings.windows125x.endsWith(
	stringToCheck := stringToTest,
	end := expectedString,
	ignoreCases := FALSE,
	trim := FALSE,
	sbcsType := Tc2_Utilities.E_SBCSType.eSBCS_CentralEuropean,
	message			:= ''
);

THIS^.AssertEquals_BOOL(
	Expected 	:= assertionIsWrong,
	Actual 		:= THIS^.assertorContainer.wasAssertionWrong,
	Message 	:= messageStringBuilder.sOut
);
END_METHOD

(*
short summary
==================
This test method tests ``assert.string.windows125x.endsWith``
method of CNM_AssertionInterfaces library with various inputs

.. <legal notes>

legal notes
=================
| SPDX-FileCopyrightText: © 2022 ekvip automation GmbH <info@ekvip.de>
| SPDX-License-Identifier: Apache-2.0
| For details check: Apache-2.0_

.. _Apache-2.0: https://www.apache.org/licenses/LICENSE-2.0

.. </legal notes>

*)


METHOD testEndsWithIgnoreCase : BOOL
VAR_INPUT
	(* for the test it's the parameter ``stringToCheck`` *)
	stringToTest 	:Tc2_System.T_MaxString;
	(* for the test it's the parameter ``end`` *)
	expectedString 	:Tc2_System.T_MaxString;
END_VAR
VAR 
	(* just the expectation if the assertion to test must be worng or true *)
	assertionIsWrong		:BOOL;
	(* contains the format string for the test message *)
	message					:Tc2_System.T_MaxString;
	(* contains ´´stringToTest´´ in upper case *)
	upperStringToTest		:Tc2_System.T_MaxString := stringToTest;
	(* contains ´´expectedString´´ in upper case *)
	upperExpectedString		:Tc2_System.T_MaxString := expectedString;
	(* used for placeholder string if stringToTest can't be printed *)
	stringToTestAsString 	:Tc2_System.T_MaxString := stringToTest;
	(* used for placeholder string if expectedString can't be printed *)
	expectedStringAsString 	:Tc2_System.T_MaxString := expectedString;
	(* TwinCAT printf with the test message *)
	messageStringBuilder	:Tc2_Utilities.FB_FormatString;
END_VAR
THIS^.assertorContainer.resetAssertor();

// both Strings to upper case
upperStringToTest := Tc2_Utilities.F_ToUCase(upperStringToTest);
upperExpectedString := Tc2_Utilities.F_ToUCase(upperExpectedString);

assertionIsWrong := ((
		Tc2_Standard.FIND(
			RIGHT(
				upperStringToTest,
				Tc2_Standard.LEN(upperExpectedString)
			), 
			upperExpectedString
			) <> 1
	) AND (
		Tc2_Standard.LEN(
			upperExpectedString
		) <> 0
	)
);

message := SEL(
	assertionIsWrong,
	'stringToCheck is $'%s$' end is $'%s$' assertion must be TRUE', 
	'stringToCheck is $'%s$' end is $'%s$' assertion must be FALSE'
);

IF (
		Tc2_Standard.LEN(stringToTest) = TO_DINT(Tc2_System.MAX_STRING_LENGTH)
) THEN
	stringToTestAsString := 'String with Tc2_System.MAX_STRING_LENGTH characters';
END_IF
IF (
		Tc2_Standard.LEN(expectedString) = TO_DINT(Tc2_System.MAX_STRING_LENGTH)
) THEN
	expectedStringAsString := 'String with Tc2_System.MAX_STRING_LENGTH characters';
END_IF

messageStringBuilder(
	sFormat := message,
	arg1 := THIS^.AnyToArg(stringToTestAsString),
	arg2 := THIS^.AnyToArg(expectedStringAsString)
);


THIS^.assertorContainer.assertor.assert.strings.windows125x.endsWith(
	stringToCheck := stringToTest,
	end := expectedString,
	ignoreCases := TRUE,
	trim := FALSE,
	message			:= ''
);

THIS^.AssertEquals_BOOL(
	Expected 	:= assertionIsWrong,
	Actual 		:= THIS^.assertorContainer.wasAssertionWrong,
	Message 	:= messageStringBuilder.sOut
);

THIS^.assertorContainer.assertor.assert.strings.windows125x.endsWith(
	stringToCheck := stringToTest,
	end := expectedString,
	ignoreCases := TRUE,
	trim := FALSE,
	sbcsType := Tc2_Utilities.E_SBCSType.eSBCS_CentralEuropean,
	message			:= ''
);

THIS^.AssertEquals_BOOL(
	Expected 	:= assertionIsWrong,
	Actual 		:= THIS^.assertorContainer.wasAssertionWrong,
	Message 	:= messageStringBuilder.sOut
);
END_METHOD

(*
short summary
==================
This test method tests ``assert.string.windows125x.endsWith``
method of CNM_AssertionInterfaces library with various inputs

.. <legal notes>

legal notes
=================
| SPDX-FileCopyrightText: © 2022 ekvip automation GmbH <info@ekvip.de>
| SPDX-License-Identifier: Apache-2.0
| For details check: Apache-2.0_

.. _Apache-2.0: https://www.apache.org/licenses/LICENSE-2.0

.. </legal notes>

*)


METHOD testEndsWithTrim : BOOL
VAR_INPUT
	(* for the test it's the parameter ``stringToCheck`` *)
	stringToTest 	:Tc2_System.T_MaxString;
	(* for the test it's the parameter ``end`` *)
	expectedString 	:Tc2_System.T_MaxString;
	(* 
	contains the expected assertion result, no calculation at runtime possible because
	CNM_UnicodeUtilities doesn't provide any functions for win125x strings and Tc2_Utilities.F_RTrim only trims spaces($20) 
	*)
	expectedAssertionResult	:BOOL;
END_VAR
VAR 
	(* just the expectation if the assertion to test must be worng or true *)
	assertionIsWrong		:BOOL;
	(* contains the format string for the test message *)
	message					:Tc2_System.T_MaxString;
	(* used for placeholder string if stringToTest can't be printed *)
	stringToTestAsString 	:Tc2_System.T_MaxString := stringToTest;
	(* used for placeholder string if expectedString can't be printed *)
	expectedStringAsString 	:Tc2_System.T_MaxString := expectedString;
	(* TwinCAT printf with the test message *)
	messageStringBuilder	:Tc2_Utilities.FB_FormatString;
END_VAR
THIS^.assertorContainer.resetAssertor();

assertionIsWrong := NOT expectedAssertionResult;

message := SEL(
	assertionIsWrong,
	'stringToCheck is $'%s$' end is $'%s$' assertion must be TRUE', 
	'stringToCheck is $'%s$' end is $'%s$' assertion must be FALSE'
);

IF (
		Tc2_Standard.LEN(stringToTest) = TO_DINT(Tc2_System.MAX_STRING_LENGTH)
) THEN
	stringToTestAsString := 'String with Tc2_System.MAX_STRING_LENGTH characters';
END_IF
IF (
		Tc2_Standard.LEN(expectedString) = TO_DINT(Tc2_System.MAX_STRING_LENGTH)
) THEN
	expectedStringAsString := 'String with Tc2_System.MAX_STRING_LENGTH characters';
END_IF

messageStringBuilder(
	sFormat := message,
	arg1 := THIS^.AnyToArg(stringToTestAsString),
	arg2 := THIS^.AnyToArg(expectedStringAsString)
);


THIS^.assertorContainer.assertor.assert.strings.windows125x.endsWith(
	stringToCheck := stringToTest,
	end := expectedString,
	ignoreCases := FALSE,
	trim := TRUE,
	message			:= ''
);

THIS^.AssertEquals_BOOL(
	Expected 	:= assertionIsWrong,
	Actual 		:= THIS^.assertorContainer.wasAssertionWrong,
	Message 	:= messageStringBuilder.sOut
);

THIS^.assertorContainer.assertor.assert.strings.windows125x.endsWith(
	stringToCheck := stringToTest,
	end := expectedString,
	ignoreCases := FALSE,
	trim := TRUE,
	sbcsType := Tc2_Utilities.E_SBCSType.eSBCS_CentralEuropean,
	message			:= ''
);

THIS^.AssertEquals_BOOL(
	Expected 	:= assertionIsWrong,
	Actual 		:= THIS^.assertorContainer.wasAssertionWrong,
	Message 	:= messageStringBuilder.sOut
);
END_METHOD

(*
short summary
==================
This test method tests ``assert.string.windows125x.isEmpty``
method of CNM_AssertionInterfaces library with various inputs

.. <legal notes>

legal notes
=================
| SPDX-FileCopyrightText: © 2022 ekvip automation GmbH <info@ekvip.de>
| SPDX-License-Identifier: Apache-2.0
| For details check: Apache-2.0_

.. _Apache-2.0: https://www.apache.org/licenses/LICENSE-2.0

.. </legal notes>

*)


METHOD testisEmpty : BOOL
VAR_INPUT
	(* for the test it's the parameter ``stringToCheck`` *)
	stringToTest	:Tc2_System.T_MaxString;
END_VAR
VAR 
	(* just the expectation if the assertion to test must be worng or true *)
	assertionIsWrong		:BOOL;
	(* contains the format string for the test message *)
	message					:Tc2_System.T_MaxString;
	(* used for placeholder string if stringToTest can't be printed *)
	stringToTestAsString 	:Tc2_System.T_MaxString := stringToTest;
	(* TwinCAT printf with the test message *)
	messageStringBuilder	:Tc2_Utilities.FB_FormatString;
END_VAR
THIS^.assertorContainer.resetAssertor();

assertionIsWrong :=  Tc2_Standard.LEN(stringToTest) > 0;

message := SEL(
	assertionIsWrong,
	'stringToCheck is $'%s$' assertion must be TRUE', 
	'stringToCheck is $'%s$' assertion must be FALSE'
);

IF (
		Tc2_Standard.LEN(stringToTest) = TO_DINT(Tc2_System.MAX_STRING_LENGTH)
) THEN
	stringToTestAsString := 'String with Tc2_System.MAX_STRING_LENGTH characters';
END_IF

messageStringBuilder(
	sFormat := message,
	arg1 := THIS^.AnyToArg(stringToTestAsString)
);

THIS^.assertorContainer.assertor.assert.strings.windows125x.isEmpty(
	stringToCheck := stringToTest,
	message			:= ''
);

THIS^.AssertEquals_BOOL(
	Expected 	:= assertionIsWrong,
	Actual 		:= THIS^.assertorContainer.wasAssertionWrong,
	Message 	:= messageStringBuilder.sOut
);
END_METHOD

(*
short summary
==================
This test method tests ``assert.string.windows125x.isEqualTo``
method of CNM_AssertionInterfaces library with various inputs

.. <legal notes>

legal notes
=================
| SPDX-FileCopyrightText: © 2022 ekvip automation GmbH <info@ekvip.de>
| SPDX-License-Identifier: Apache-2.0
| For details check: Apache-2.0_

.. _Apache-2.0: https://www.apache.org/licenses/LICENSE-2.0

.. </legal notes>

*)


METHOD testIsEqualTo : BOOL
VAR_INPUT
	(* for the test it's the parameter ``stringToCheck`` *)
	stringToTest 	:Tc2_System.T_MaxString;
	(* for the test it's the parameter ``expected`` *)
	expectedString 	:Tc2_System.T_MaxString;
END_VAR
VAR 
	(* just the expectation if the assertion to test must be worng or true *)
	assertionIsWrong		:BOOL;
	(* contains the format string for the test message *)
	message					:Tc2_System.T_MaxString;
	(* used for placeholder string if stringToTest can't be printed *)
	stringToTestAsString 	:Tc2_System.T_MaxString := stringToTest;
	(* used for placeholder string if expectedString can't be printed *)
	expectedStringAsString 	:Tc2_System.T_MaxString := expectedString;
	(* TwinCAT printf with the test message *)
	messageStringBuilder	:Tc2_Utilities.FB_FormatString;
END_VAR
THIS^.assertorContainer.resetAssertor();

assertionIsWrong := ((
		Tc2_Standard.LEN(
			stringToTest
		) <> Tc2_Standard.LEN(expectedString)
	) OR_ELSE (
		Tc2_Standard.FIND(
			stringToTest,
			expectedString
		) <> 1
	) AND (
		Tc2_Standard.LEN(stringToTest) <> 0
	)
);

message := SEL(
	assertionIsWrong,
	'stringToCheck is $'%s$' expected is $'%s$' assertion must be TRUE', 
	'stringToCheck is $'%s$' expected is $'%s$' assertion must be FALSE'
);

IF (
		Tc2_Standard.LEN(stringToTest) = TO_DINT(Tc2_System.MAX_STRING_LENGTH)
) THEN
	stringToTestAsString := 'String with Tc2_System.MAX_STRING_LENGTH characters';
END_IF
IF (
		Tc2_Standard.LEN(expectedString) = TO_DINT(Tc2_System.MAX_STRING_LENGTH)
) THEN
	expectedStringAsString := 'String with Tc2_System.MAX_STRING_LENGTH characters';
END_IF

messageStringBuilder(
	sFormat := message,
	arg1 := THIS^.AnyToArg(stringToTestAsString),
	arg2 := THIS^.AnyToArg(expectedStringAsString)
);

THIS^.assertorContainer.assertor.assert.strings.windows125x.isEqualTo(
	stringToCheck := stringToTest,
	expected := expectedString,
	ignoreCases := FALSE,
	message			:= ''
);

THIS^.AssertEquals_BOOL(
	Expected 	:= assertionIsWrong,
	Actual 		:= THIS^.assertorContainer.wasAssertionWrong,
	Message 	:= messageStringBuilder.sOut
);

THIS^.assertorContainer.assertor.assert.strings.windows125x.isEqualTo(
	stringToCheck := stringToTest,
	expected := expectedString,
	ignoreCases := FALSE,
	sbcsType := Tc2_Utilities.E_SBCSType.eSBCS_CentralEuropean,
	message			:= ''
);

THIS^.AssertEquals_BOOL(
	Expected 	:= assertionIsWrong,
	Actual 		:= THIS^.assertorContainer.wasAssertionWrong,
	Message 	:= messageStringBuilder.sOut
);
END_METHOD

(*
short summary
==================
This test method tests ``assert.string.windows125x.isEqualTo``
method of CNM_AssertionInterfaces library with various inputs

.. <legal notes>

legal notes
=================
| SPDX-FileCopyrightText: © 2022 ekvip automation GmbH <info@ekvip.de>
| SPDX-License-Identifier: Apache-2.0
| For details check: Apache-2.0_

.. _Apache-2.0: https://www.apache.org/licenses/LICENSE-2.0

.. </legal notes>

*)


METHOD testIsEqualToIgnoreCase : BOOL
VAR_INPUT
	(* for the test it's the parameter ``stringToCheck`` *)
	stringToTest 	:Tc2_System.T_MaxString;
	(* for the test it's the parameter ``expected`` *)
	expectedString 	:Tc2_System.T_MaxString;
END_VAR
VAR 
	(* just the expectation if the assertion to test must be worng or true *)
	assertionIsWrong		:BOOL;
	(* contains the format string for the test message *)
	message					:Tc2_System.T_MaxString;
	(* contains ´´stringToTest´´ in upper case *)
	upperStringToTest		:Tc2_System.T_MaxString := stringToTest;
	(* contains ´´expectedString´´ in upper case *)
	upperExpectedString		:Tc2_System.T_MaxString := expectedString;
	(* used for placeholder string if stringToTest can't be printed *)
	stringToTestAsString 	:Tc2_System.T_MaxString := stringToTest;
	(* used for placeholder string if expectedString can't be printed *)
	expectedStringAsString 	:Tc2_System.T_MaxString := expectedString;
	(* TwinCAT printf with the test message *)
	messageStringBuilder	:Tc2_Utilities.FB_FormatString;
END_VAR
THIS^.assertorContainer.resetAssertor();

// both Strings to upper case
upperStringToTest := Tc2_Utilities.F_ToUCase(upperStringToTest);
upperExpectedString := Tc2_Utilities.F_ToUCase(upperExpectedString);

assertionIsWrong := ((
		Tc2_Standard.LEN(
			upperStringToTest
		) <> Tc2_Standard.LEN(upperExpectedString)				
	) OR (
		Tc2_Standard.FIND(
			upperStringToTest,
			upperExpectedString
		) <> 1
	) AND (
		Tc2_Standard.LEN(upperStringToTest) <> 0
	)
);

message := SEL(
	assertionIsWrong,
	'stringToCheck is $'%s$' expected is $'%s$' assertion must be TRUE', 
	'stringToCheck is $'%s$' expected is $'%s$' assertion must be FALSE'
);

IF (
		Tc2_Standard.LEN(stringToTest) = TO_DINT(Tc2_System.MAX_STRING_LENGTH)
) THEN
	stringToTestAsString := 'String with Tc2_System.MAX_STRING_LENGTH characters';
END_IF
IF (
		Tc2_Standard.LEN(expectedString) = TO_DINT(Tc2_System.MAX_STRING_LENGTH)
) THEN
	expectedStringAsString := 'String with Tc2_System.MAX_STRING_LENGTH characters';
END_IF

messageStringBuilder(
	sFormat := message,
	arg1 := THIS^.AnyToArg(stringToTestAsString),
	arg2 := THIS^.AnyToArg(expectedStringAsString)
);


THIS^.assertorContainer.assertor.assert.strings.windows125x.isEqualTo(
	stringToCheck := stringToTest,
	expected := expectedString,
	ignoreCases := TRUE,
	message			:= ''
);

THIS^.AssertEquals_BOOL(
	Expected 	:= assertionIsWrong,
	Actual 		:= THIS^.assertorContainer.wasAssertionWrong,
	Message 	:= messageStringBuilder.sOut
);

THIS^.assertorContainer.assertor.assert.strings.windows125x.isEqualTo(
	stringToCheck := stringToTest,
	expected := expectedString,
	ignoreCases := TRUE,
	sbcsType := Tc2_Utilities.E_SBCSType.eSBCS_CentralEuropean,
	message			:= ''
);

THIS^.AssertEquals_BOOL(
	Expected 	:= assertionIsWrong,
	Actual 		:= THIS^.assertorContainer.wasAssertionWrong,
	Message 	:= messageStringBuilder.sOut
);
END_METHOD

(*
short summary
==================
This test method tests ``assert.string.windows125x.isNotEmpty``
method of CNM_AssertionInterfaces library with various inputs

.. <legal notes>

legal notes
=================
| SPDX-FileCopyrightText: © 2022 ekvip automation GmbH <info@ekvip.de>
| SPDX-License-Identifier: Apache-2.0
| For details check: Apache-2.0_

.. _Apache-2.0: https://www.apache.org/licenses/LICENSE-2.0

.. </legal notes>

*)


METHOD testIsNotEmpty : BOOL
VAR_INPUT
	(* for the test it's the parameter ``stringToCheck`` *)
	stringToTest	:Tc2_System.T_MaxString;
END_VAR
VAR 
	(* just the expectation if the assertion to test must be worng or true *)
	assertionIsWrong		:BOOL;
	(* contains the format string for the test message *)
	message					:Tc2_System.T_MaxString;
	(* used for placeholder string if stringToTest can't be printed *)
	stringToTestAsString 	:Tc2_System.T_MaxString := stringToTest;
	(* TwinCAT printf with the test message *)
	messageStringBuilder	:Tc2_Utilities.FB_FormatString;
END_VAR
THIS^.assertorContainer.resetAssertor();

assertionIsWrong :=  Tc2_Standard.LEN(stringToTest) = 0;

message := SEL(
	assertionIsWrong,
	'stringToCheck is $'%s$' assertion must be TRUE', 
	'stringToCheck is $'%s$' assertion must be FALSE'
);

IF (
		Tc2_Standard.LEN(stringToTest) = TO_DINT(Tc2_System.MAX_STRING_LENGTH)
) THEN
	stringToTestAsString := 'String with Tc2_System.MAX_STRING_LENGTH characters';
END_IF

messageStringBuilder(
	sFormat := message,
	arg1 := THIS^.AnyToArg(stringToTestAsString)
);


THIS^.assertorContainer.assertor.assert.strings.windows125x.isNotEmpty(
	stringToCheck := stringToTest,
	message			:= ''
);

THIS^.AssertEquals_BOOL(
	Expected 	:= assertionIsWrong,
	Actual 		:= THIS^.assertorContainer.wasAssertionWrong,
	Message 	:= messageStringBuilder.sOut
);
END_METHOD

(*
short summary
==================
This test method tests ``assert.string.utf8.isNotEqualTo``
method of CNM_AssertionInterfaces library with various inputs

.. <legal notes>

legal notes
=================
| SPDX-FileCopyrightText: © 2022 ekvip automation GmbH <info@ekvip.de>
| SPDX-License-Identifier: Apache-2.0
| For details check: Apache-2.0_

.. _Apache-2.0: https://www.apache.org/licenses/LICENSE-2.0

.. </legal notes>

*)


METHOD testIsNotEqualTo : BOOL
VAR_INPUT
	(* for the test it's the parameter ``stringToCheck`` *)
	stringToTest 	:Tc2_System.T_MaxString;
	(* for the test it's the parameter ``unexpected`` *)
	expectedString 	:Tc2_System.T_MaxString;
END_VAR
VAR 
	(* just the expectation if the assertion to test must be worng or true *)
	assertionIsWrong		:BOOL;
	(* contains the format string for the test message *)
	message					:Tc2_System.T_MaxString;
	(* used for placeholder string if stringToTest can't be printed *)
	stringToTestAsString 	:Tc2_System.T_MaxString := stringToTest;
	(* used for placeholder string if expectedString can't be printed *)
	expectedStringAsString 	:Tc2_System.T_MaxString := expectedString;
	(* TwinCAT printf with the test message *)
	messageStringBuilder	:Tc2_Utilities.FB_FormatString;
END_VAR
THIS^.assertorContainer.resetAssertor();

assertionIsWrong := (stringToTest = expectedString);

message := SEL(
	assertionIsWrong,
	'stringToCheck is $'%s$' unexpected is $'%s$' assertion must be TRUE', 
	'stringToCheck is $'%s$' unexpected is $'%s$' assertion must be FALSE'
);

IF (
		Tc2_Standard.LEN(stringToTest) = TO_UINT(Tc2_System.MAX_STRING_LENGTH)
) THEN
	stringToTestAsString := 'String with Tc2_System.MAX_STRING_LENGTH characters';
END_IF
IF (
		Tc2_Standard.LEN(expectedString) = TO_UINT(Tc2_System.MAX_STRING_LENGTH)
) THEN
	expectedStringAsString := 'String with Tc2_System.MAX_STRING_LENGTH characters';
END_IF

messageStringBuilder(
	sFormat := message,
	arg1 := THIS^.AnyToArg(stringToTestAsString),
	arg2 := THIS^.AnyToArg(expectedStringAsString)
);


THIS^.assertorContainer.assertor.assert.strings.windows125x.isNotEqualTo(
	stringToCheck := stringToTest,
	unexpected := expectedString,
	ignoreCases := FALSE,
	message			:= ''
);

THIS^.AssertEquals_BOOL(
	Expected 	:= assertionIsWrong,
	Actual 		:= THIS^.assertorContainer.wasAssertionWrong,
	Message 	:= messageStringBuilder.sOut
);

THIS^.assertorContainer.assertor.assert.strings.windows125x.isNotEqualTo(
	stringToCheck := stringToTest,
	unexpected := expectedString,
	ignoreCases := FALSE,
	sbcsType := Tc2_Utilities.E_SBCSType.eSBCS_CentralEuropean,
	message			:= ''
);

THIS^.AssertEquals_BOOL(
	Expected 	:= assertionIsWrong,
	Actual 		:= THIS^.assertorContainer.wasAssertionWrong,
	Message 	:= messageStringBuilder.sOut
);
END_METHOD

(*
short summary
==================
This test method tests ``assert.string.utf8.isNotEqualTo``
method of CNM_AssertionInterfaces library with various inputs

.. <legal notes>

legal notes
=================
| SPDX-FileCopyrightText: © 2022 ekvip automation GmbH <info@ekvip.de>
| SPDX-License-Identifier: Apache-2.0
| For details check: Apache-2.0_

.. _Apache-2.0: https://www.apache.org/licenses/LICENSE-2.0

.. </legal notes>

*)


METHOD testIsNotEqualToIgnoreCase : BOOL
VAR_INPUT
	(* for the test it's the parameter ``stringToCheck`` *)
	stringToTest 	:Tc2_System.T_MaxString;
	(* for the test it's the parameter ``unexpected`` *)
	expectedString 	:Tc2_System.T_MaxString;
END_VAR
VAR 
	(* just the expectation if the assertion to test must be worng or true *)
	assertionIsWrong		:BOOL;
	(* contains the format string for the test message *)
	message					:Tc2_System.T_MaxString;
	(* contains ´´stringToTest´´ in upper case *)
	upperStringToTest		:Tc2_System.T_MaxString := stringToTest;
	(* contains ´´expectedString´´ in upper case *)
	upperExpectedString		:Tc2_System.T_MaxString := expectedString;
	(* used for placeholder string if stringToTest can't be printed *)
	stringToTestAsString 	:Tc2_System.T_MaxString := stringToTest;
	(* used for placeholder string if expectedString can't be printed *)
	expectedStringAsString	:Tc2_System.T_MaxString := expectedString;
	(* TwinCAT printf with the test message *)
	messageStringBuilder	:Tc2_Utilities.FB_FormatString;
END_VAR
THIS^.assertorContainer.resetAssertor();

// both Strings to upper case
upperStringToTest := Tc2_Utilities.F_ToUCase(upperStringToTest);
upperExpectedString := Tc2_Utilities.F_ToUCase(upperExpectedString);

assertionIsWrong := (stringToTest = expectedString);

message := SEL(
	assertionIsWrong,
	'stringToCheck is $'%s$' unexpected is $'%s$' assertion must be TRUE', 
	'stringToCheck is $'%s$' unexpected is $'%s$' assertion must be FALSE'
);

IF (
		Tc2_Standard.LEN(stringToTest) = TO_DINT(Tc2_System.MAX_STRING_LENGTH)
) THEN
	stringToTestAsString := 'String with Tc2_System.MAX_STRING_LENGTH characters';
END_IF
IF (
		Tc2_Standard.LEN(expectedString) = TO_DINT(Tc2_System.MAX_STRING_LENGTH)
) THEN
	expectedStringAsString := 'String with Tc2_System.MAX_STRING_LENGTH characters';
END_IF

messageStringBuilder(
	sFormat := message,
	arg1 := THIS^.AnyToArg(stringToTestAsString),
	arg2 := THIS^.AnyToArg(expectedStringAsString)
);


THIS^.assertorContainer.assertor.assert.strings.windows125x.isNotEqualTo(
	stringToCheck := stringToTest,
	unexpected := expectedString,
	ignoreCases := TRUE,
	message			:= ''
);

THIS^.AssertEquals_BOOL(
	Expected 	:= assertionIsWrong,
	Actual 		:= THIS^.assertorContainer.wasAssertionWrong,
	Message 	:= messageStringBuilder.sOut
);

THIS^.assertorContainer.assertor.assert.strings.windows125x.isNotEqualTo(
	stringToCheck := stringToTest,
	unexpected := expectedString,
	ignoreCases := TRUE,
	sbcsType := Tc2_Utilities.E_SBCSType.eSBCS_CentralEuropean,
	message			:= ''
);

THIS^.AssertEquals_BOOL(
	Expected 	:= assertionIsWrong,
	Actual 		:= THIS^.assertorContainer.wasAssertionWrong,
	Message 	:= messageStringBuilder.sOut
);
END_METHOD

(*
short summary
==================
This test method tests ``assert.string.windows125x.lengthIsBetween``
method of CNM_AssertionInterfaces library with various inputs

.. <legal notes>

legal notes
=================
| SPDX-FileCopyrightText: © 2022 ekvip automation GmbH <info@ekvip.de>
| SPDX-License-Identifier: Apache-2.0
| For details check: Apache-2.0_

.. _Apache-2.0: https://www.apache.org/licenses/LICENSE-2.0

.. </legal notes>

*)


METHOD testLengthIsBetween : BOOL
VAR_INPUT
	(* for the test it's the parameter ``stringToCheck`` *)
	stringToTest	:Tc2_System.T_MaxString;
	(* for the test it's the parameter ``maxLength`` *)
	maxLength 		:USINT;
	(* for the test it's the parameter ``minLength`` *)
	minLength 		:USINT;
END_VAR
VAR 
	(* just the expectation if the assertion to test must be worng or true *)
	assertionIsWrong		:BOOL;
	(* contains the format string for the test message *)
	message					:Tc2_System.T_MaxString;
	(* used for placeholder string if stringToTest can't be printed *)
	stringToTestAsString 	:Tc2_System.T_MaxString := stringToTest;
	(* TwinCAT printf with the test message *)
	messageStringBuilder	:Tc2_Utilities.FB_FormatString;
END_VAR
THIS^.assertorContainer.resetAssertor();

assertionIsWrong := ((
		Tc2_Standard.LEN(
			stringToTest
		) < minLength
	) OR_ELSE (
		Tc2_Standard.LEN(
			stringToTest
		) > maxLength
	)
);

message := SEL(
	assertionIsWrong,
	'stringToCheck is $'%s$' with maxLength %u and minLength %u assertion must be TRUE', 
	'stringToCheck is $'%s$' with maxLength %u and minLength %u assertion must be FALSE'
);

IF (
		Tc2_Standard.LEN(stringToTest) = TO_DINT(Tc2_System.MAX_STRING_LENGTH)
) THEN
	stringToTestAsString := 'String with Tc2_System.MAX_STRING_LENGTH characters';
END_IF


messageStringBuilder(
	sFormat := message,
	arg1 := THIS^.AnyToArg(stringToTestAsString),
	arg2 := THIS^.AnyToArg(maxLength),
	arg3 := THIS^.AnyToArg(minLength)
);


THIS^.assertorContainer.assertor.assert.strings.windows125x.lengthIsBetween(
	stringToCheck := stringToTest,
	maxLength := maxLength,
	minLength := minLength,
	message			:= ''
);

THIS^.AssertEquals_BOOL(
	Expected 	:= assertionIsWrong,
	Actual 		:= THIS^.assertorContainer.wasAssertionWrong,
	Message 	:= messageStringBuilder.sOut
);
END_METHOD

(*
short summary
==================
This test method tests ``assert.string.windows125x.lengthIsExact``
method of CNM_AssertionInterfaces library with various inputs

.. <legal notes>

legal notes
=================
| SPDX-FileCopyrightText: © 2022 ekvip automation GmbH <info@ekvip.de>
| SPDX-License-Identifier: Apache-2.0
| For details check: Apache-2.0_

.. _Apache-2.0: https://www.apache.org/licenses/LICENSE-2.0

.. </legal notes>

*)

METHOD testLengthIsExact : BOOL
VAR_INPUT
	(* for the test it's the parameter ``stringToCheck`` *)
	stringToTest	:Tc2_System.T_MaxString;
	(* for the test it's the parameter ``expectedLength`` *)
	expectedLength	:USINT;
END_VAR
VAR 
	(* just the expectation if the assertion to test must be worng or true *)
	assertionIsWrong		:BOOL;
	(* contains the format string for the test message *)
	message					:Tc2_System.T_MaxString;
	(* used for placeholder string if stringToTest can't be printed *)
	stringToTestAsString 	:Tc2_System.T_MaxString := stringToTest;
	(* TwinCAT printf with the test message *)
	messageStringBuilder	:Tc2_Utilities.FB_FormatString;
END_VAR
THIS^.assertorContainer.resetAssertor();

assertionIsWrong := Tc2_Standard.LEN(stringToTest) <> expectedLength;

message := SEL(
	assertionIsWrong,
	'stringToCheck is $'%s$' expectedLength is %u assertion must be TRUE', 
	'stringToCheck is $'%s$' expectedLength is %u assertion must be FALSE'
);

IF (
		Tc2_Standard.LEN(stringToTest) = TO_DINT(Tc2_System.MAX_STRING_LENGTH)
) THEN
	stringToTestAsString := 'String with Tc2_System.MAX_STRING_LENGTH characters';
END_IF

messageStringBuilder(
	sFormat := message,
	arg1 := THIS^.AnyToArg(stringToTestAsString),
	arg2 := THIS^.AnyToArg(expectedLength),
);


THIS^.assertorContainer.assertor.assert.strings.windows125x.lengthIsExact(
	stringToCheck := stringToTest,
	expectedLength := expectedLength,
	message			:= ''
);

THIS^.AssertEquals_BOOL(
	Expected 	:= assertionIsWrong,
	Actual 		:= THIS^.assertorContainer.wasAssertionWrong,
	Message 	:= messageStringBuilder.sOut
);
END_METHOD

(*
short summary
==================
This test method tests ``assert.string.windows125x.lengthIsMax``
method of CNM_AssertionInterfaces library with various inputs

.. <legal notes>

legal notes
=================
| SPDX-FileCopyrightText: © 2022 ekvip automation GmbH <info@ekvip.de>
| SPDX-License-Identifier: Apache-2.0
| For details check: Apache-2.0_

.. _Apache-2.0: https://www.apache.org/licenses/LICENSE-2.0

.. </legal notes>

*)


METHOD testLengthIsMax : BOOL
VAR_INPUT
	(* for the test it's the parameter ``stringToCheck`` *)
	stringToTest	:Tc2_System.T_MaxString;
	(* for the test it's the parameter ``maxLength`` *)
	expectedLength	:USINT;
END_VAR
VAR 
	(* just the expectation if the assertion to test must be worng or true *)
	assertionIsWrong		:BOOL;
	(* contains the format string for the test message *)
	message					:Tc2_System.T_MaxString;
	(* used for placeholder string if stringToTest can't be printed *)
	stringToTestAsString 	:Tc2_System.T_MaxString := stringToTest;
	(* TwinCAT printf with the test message *)
	messageStringBuilder	:Tc2_Utilities.FB_FormatString;
END_VAR
THIS^.assertorContainer.resetAssertor();

assertionIsWrong := Tc2_Standard.LEN(stringToTest) > expectedLength;

message := SEL(
	assertionIsWrong,
	'stringToCheck is $'%s$' maxLength is %u assertion must be TRUE', 
	'stringToCheck is $'%s$' maxLength is %u assertion must be FALSE'
);

IF (
		Tc2_Standard.LEN(stringToTest) = TO_DINT(Tc2_System.MAX_STRING_LENGTH)
) THEN
	stringToTestAsString := 'String with Tc2_System.MAX_STRING_LENGTH characters';
END_IF

messageStringBuilder(
	sFormat := message,
	arg1 := THIS^.AnyToArg(stringToTestAsString),
	arg2 := THIS^.AnyToArg(expectedLength),
);


THIS^.assertorContainer.assertor.assert.strings.windows125x.lengthIsMax(
	stringToCheck := stringToTest,
	maxLength := expectedLength,
	message			:= ''
);

THIS^.AssertEquals_BOOL(
	Expected 	:= assertionIsWrong,
	Actual 		:= THIS^.assertorContainer.wasAssertionWrong,
	Message 	:= messageStringBuilder.sOut
);
END_METHOD

(*
short summary
==================
This test method tests ``assert.string.windows125x.lengthIsMin``
method of CNM_AssertionInterfaces library with various inputs

.. <legal notes>

legal notes
=================
| SPDX-FileCopyrightText: © 2022 ekvip automation GmbH <info@ekvip.de>
| SPDX-License-Identifier: Apache-2.0
| For details check: Apache-2.0_

.. _Apache-2.0: https://www.apache.org/licenses/LICENSE-2.0

.. </legal notes>

*)


METHOD testLengthIsMin : BOOL
VAR_INPUT
	(* for the test it's the parameter ``stringToCheck`` *)
	stringToTest	:Tc2_System.T_MaxString;
	(* for the test it's the parameter ``minLength`` *)
	expectedLength	:USINT;
END_VAR
VAR 
	(* just the expectation if the assertion to test must be worng or true *)
	assertionIsWrong		:BOOL;
	(* contains the format string for the test message *)
	message					:Tc2_System.T_MaxString;
	(* used for placeholder string if stringToTest can't be printed *)
	stringToTestAsString 	:Tc2_System.T_MaxString := stringToTest;
	(* TwinCAT printf with the test message *)
	messageStringBuilder	:Tc2_Utilities.FB_FormatString;
END_VAR
THIS^.assertorContainer.resetAssertor();

assertionIsWrong := Tc2_Standard.LEN(stringToTest) < expectedLength;

message := SEL(
	assertionIsWrong,
	'stringToCheck is $'%s$' minLength is %u assertion must be TRUE', 
	'stringToCheck is $'%s$' minLength is %u assertion must be FALSE'
);

IF (
		Tc2_Standard.LEN(stringToTest) = TO_DINT(Tc2_System.MAX_STRING_LENGTH)
) THEN
	stringToTestAsString := 'String with Tc2_System.MAX_STRING_LENGTH characters';
END_IF

messageStringBuilder(
	sFormat := message,
	arg1 := THIS^.AnyToArg(stringToTestAsString),
	arg2 := THIS^.AnyToArg(expectedLength),
);


THIS^.assertorContainer.assertor.assert.strings.windows125x.lengthIsMin(
	stringToCheck := stringToTest,
	minLength := expectedLength,
	message			:= ''
);

THIS^.AssertEquals_BOOL(
	Expected 	:= assertionIsWrong,
	Actual 		:= THIS^.assertorContainer.wasAssertionWrong,
	Message 	:= messageStringBuilder.sOut
);
END_METHOD

(*
short summary
==================
This test method tests ``assert.string.windows125x.startsWith``
method of CNM_AssertionInterfaces library with various inputs

.. <legal notes>

legal notes
=================
| SPDX-FileCopyrightText: © 2022 ekvip automation GmbH <info@ekvip.de>
| SPDX-License-Identifier: Apache-2.0
| For details check: Apache-2.0_

.. _Apache-2.0: https://www.apache.org/licenses/LICENSE-2.0

.. </legal notes>

*)


METHOD testStartsWith : BOOL
VAR_INPUT
	(* for the test it's the parameter ``stringToCheck`` *)
	stringToTest 	:Tc2_System.T_MaxString;
	(* for the test it's the parameter ``end`` *)
	expectedString 	:Tc2_System.T_MaxString;
END_VAR
VAR 
	(* just the expectation if the assertion to test must be worng or true *)
	assertionIsWrong		:BOOL;
	(* contains the format string for the test message *)
	message					:Tc2_System.T_MaxString;
	(* used for placeholder string if stringToTest can't be printed *)
	stringToTestAsString 	:Tc2_System.T_MaxString := stringToTest;
	(* used for placeholder string if expectedString can't be printed *)
	expectedStringAsString 	:Tc2_System.T_MaxString := expectedString;
	(* TwinCAT printf with the test message *)
	messageStringBuilder	:Tc2_Utilities.FB_FormatString;
END_VAR
THIS^.assertorContainer.resetAssertor();

assertionIsWrong := ((
		Tc2_Standard.FIND(
			stringToTest,
			expectedString
		) <> 1
	) AND (
		Tc2_Standard.LEN(
			expectedString
		) <> 0
	)
);

message := SEL(
	assertionIsWrong,
	'stringToCheck is $'%s$' end is $'%s$' assertion must be TRUE', 
	'stringToCheck is $'%s$' end is $'%s$' assertion must be FALSE'
);

IF (
		Tc2_Standard.LEN(stringToTest) = TO_DINT(Tc2_System.MAX_STRING_LENGTH)
) THEN
	stringToTestAsString := 'String with Tc2_System.MAX_STRING_LENGTH characters';
END_IF
IF (
		Tc2_Standard.LEN(expectedString) = TO_DINT(Tc2_System.MAX_STRING_LENGTH)
) THEN
	expectedStringAsString := 'String with Tc2_System.MAX_STRING_LENGTH characters';
END_IF

messageStringBuilder(
	sFormat := message,
	arg1 := THIS^.AnyToArg(stringToTestAsString),
	arg2 := THIS^.AnyToArg(expectedStringAsString)
);


THIS^.assertorContainer.assertor.assert.strings.windows125x.startsWith(
	stringToCheck := stringToTest,
	start := expectedString,
	ignoreCases := FALSE,
	trim := FALSE,
	message			:= ''
);

THIS^.AssertEquals_BOOL(
	Expected 	:= assertionIsWrong,
	Actual 		:= THIS^.assertorContainer.wasAssertionWrong,
	Message 	:= messageStringBuilder.sOut
);

THIS^.assertorContainer.assertor.assert.strings.windows125x.startsWith(
	stringToCheck := stringToTest,
	start := expectedString,
	ignoreCases := FALSE,
	trim := FALSE,
	sbcsType := Tc2_Utilities.E_SBCSType.eSBCS_CentralEuropean,
	message			:= ''
);

THIS^.AssertEquals_BOOL(
	Expected 	:= assertionIsWrong,
	Actual 		:= THIS^.assertorContainer.wasAssertionWrong,
	Message 	:= messageStringBuilder.sOut
);
END_METHOD

(*
short summary
==================
This test method tests ``assert.string.windows125x.startsWith``
method of CNM_AssertionInterfaces library with various inputs

.. <legal notes>

legal notes
=================
| SPDX-FileCopyrightText: © 2022 ekvip automation GmbH <info@ekvip.de>
| SPDX-License-Identifier: Apache-2.0
| For details check: Apache-2.0_

.. _Apache-2.0: https://www.apache.org/licenses/LICENSE-2.0

.. </legal notes>

*)


METHOD testStartsWithIgnoreCase : BOOL
VAR_INPUT
	(* for the test it's the parameter ``stringToCheck`` *)
	stringToTest	:Tc2_System.T_MaxString;
	(* for the test it's the parameter ``end`` *)
	expectedString	:Tc2_System.T_MaxString;
END_VAR
VAR 
	(* just the expectation if the assertion to test must be worng or true *)
	assertionIsWrong		:BOOL;
	(* contains the format string for the test message *)
	message					:Tc2_System.T_MaxString;
	(* contains ´´stringToTest´´ in upper case *)
	upperStringToTest		:Tc2_System.T_MaxString := stringToTest;
	(* contains ´´expectedString´´ in upper case *)
	upperExpectedString		:Tc2_System.T_MaxString := expectedString;
	(* used for placeholder string if stringToTest can't be printed *)
	stringToTestAsString 	:Tc2_System.T_MaxString := stringToTest;
	(* used for placeholder string if expectedString can't be printed *)
	expectedStringAsString 	:Tc2_System.T_MaxString := expectedString;
	(* TwinCAT printf with the test message *)
	messageStringBuilder	:Tc2_Utilities.FB_FormatString;
END_VAR
THIS^.assertorContainer.resetAssertor();

// both Strings to upper case
upperStringToTest := Tc2_Utilities.F_ToUCase(upperStringToTest);
upperExpectedString := Tc2_Utilities.F_ToUCase(upperExpectedString);

assertionIsWrong := ((
		Tc2_Standard.FIND(
			upperStringToTest,
			upperExpectedString
		) <> 1
	) AND (
		Tc2_Standard.LEN(
			upperExpectedString
		) <> 0
	)
);

message := SEL(
	assertionIsWrong,
	'stringToCheck is $'%s$' end is $'%s$' assertion must be TRUE', 
	'stringToCheck is $'%s$' end is $'%s$' assertion must be FALSE'
);

IF (
		Tc2_Standard.LEN(stringToTest) = TO_DINT(Tc2_System.MAX_STRING_LENGTH)
) THEN
	stringToTestAsString := 'String with Tc2_System.MAX_STRING_LENGTH characters';
END_IF
IF (
		Tc2_Standard.LEN(expectedString) = TO_DINT(Tc2_System.MAX_STRING_LENGTH)
) THEN
	expectedStringAsString := 'String with Tc2_System.MAX_STRING_LENGTH characters';
END_IF

messageStringBuilder(
	sFormat := message,
	arg1 := THIS^.AnyToArg(stringToTestAsString),
	arg2 := THIS^.AnyToArg(expectedStringAsString)
);


THIS^.assertorContainer.assertor.assert.strings.windows125x.startsWith(
	stringToCheck := stringToTest,
	start := expectedString,
	ignoreCases := TRUE,
	trim := FALSE,
	message			:= ''
);

THIS^.AssertEquals_BOOL(
	Expected 	:= assertionIsWrong,
	Actual 		:= THIS^.assertorContainer.wasAssertionWrong,
	Message 	:= messageStringBuilder.sOut
);

THIS^.assertorContainer.assertor.assert.strings.windows125x.startsWith(
	stringToCheck := stringToTest,
	start := expectedString,
	ignoreCases := TRUE,
	trim := FALSE,
	sbcsType := Tc2_Utilities.E_SBCSType.eSBCS_CentralEuropean,
	message			:= ''
);

THIS^.AssertEquals_BOOL(
	Expected 	:= assertionIsWrong,
	Actual 		:= THIS^.assertorContainer.wasAssertionWrong,
	Message 	:= messageStringBuilder.sOut
);
END_METHOD

(*
short summary
==================
This test method tests ``assert.string.windows125x.startsWith``
method of CNM_AssertionInterfaces library with various inputs

.. <legal notes>

legal notes
=================
| SPDX-FileCopyrightText: © 2022 ekvip automation GmbH <info@ekvip.de>
| SPDX-License-Identifier: Apache-2.0
| For details check: Apache-2.0_

.. _Apache-2.0: https://www.apache.org/licenses/LICENSE-2.0

.. </legal notes>

*)


METHOD testStartsWithTrim : BOOL
VAR_INPUT
	(* for the test it's the parameter ``stringToCheck`` *)
	stringToTest 			:Tc2_System.T_MaxString;
	(* for the test it's the parameter ``end`` *)
	expectedString			:Tc2_System.T_MaxString;
	(* 
	contains the expected assertion result, no calculation at runtime possible because
	CNM_UnicodeUtilities doesn't provide any functions for win125x strings and Tc2_Utilities.F_RTrim only trims spaces($20) 
	*)
	expectedAssertionResult	:BOOL;
END_VAR
VAR 
	(* just the expectation if the assertion to test must be worng or true *)
	assertionIsWrong		:BOOL;
	(* contains the format string for the test message *)
	message					:Tc2_System.T_MaxString;
	(* used for placeholder string if stringToTest can't be printed *)
	stringToTestAsString 	:Tc2_System.T_MaxString := stringToTest;
	(* used for placeholder string if expectedString can't be printed *)
	expectedStringAsString 	:Tc2_System.T_MaxString := expectedString;
	(* TwinCAT printf with the test message *)
	messageStringBuilder	:Tc2_Utilities.FB_FormatString;
END_VAR
THIS^.assertorContainer.resetAssertor();

assertionIsWrong := NOT expectedAssertionResult;

message := SEL(
	assertionIsWrong,
	'stringToCheck is $'%s$' end is $'%s$' assertion must be TRUE', 
	'stringToCheck is $'%s$' end is $'%s$' assertion must be FALSE'
);

IF (
		Tc2_Standard.LEN(stringToTest) = TO_DINT(Tc2_System.MAX_STRING_LENGTH)
) THEN
	stringToTestAsString := 'String with Tc2_System.MAX_STRING_LENGTH characters';
END_IF
IF (
		Tc2_Standard.LEN(expectedString) = TO_DINT(Tc2_System.MAX_STRING_LENGTH)
) THEN
	expectedStringAsString := 'String with Tc2_System.MAX_STRING_LENGTH characters';
END_IF

messageStringBuilder(
	sFormat := message,
	arg1 := THIS^.AnyToArg(stringToTestAsString),
	arg2 := THIS^.AnyToArg(expectedStringAsString)
);


THIS^.assertorContainer.assertor.assert.strings.windows125x.startsWith(
	stringToCheck := stringToTest,
	start := expectedString,
	ignoreCases := FALSE,
	trim := TRUE,
	message			:= ''
);

THIS^.AssertEquals_BOOL(
	Expected 	:= assertionIsWrong,
	Actual 		:= THIS^.assertorContainer.wasAssertionWrong,
	Message 	:= messageStringBuilder.sOut
);

THIS^.assertorContainer.assertor.assert.strings.windows125x.startsWith(
	stringToCheck := stringToTest,
	start := expectedString,
	ignoreCases := FALSE,
	trim := TRUE,
	sbcsType := Tc2_Utilities.E_SBCSType.eSBCS_CentralEuropean,
	message			:= ''
);

THIS^.AssertEquals_BOOL(
	Expected 	:= assertionIsWrong,
	Actual 		:= THIS^.assertorContainer.wasAssertionWrong,
	Message 	:= messageStringBuilder.sOut
);
END_METHOD

END_FUNCTION_BLOCK

// ---- AssertionTester/AssertionTests/TimeAssertions/classes/LTimeAssertionsTests.TcPOU
(*

short summary
==================
This class tests all methods of LTIME assertions
with various combinations of inputs and checks expected 
outputs are satisfied or not

.. <legal notes>

legal notes
=================
| SPDX-FileCopyrightText: © 2022 ekvip automation GmbH <info@ekvip.de>
| SPDX-License-Identifier: Apache-2.0
| For details check: Apache-2.0_

.. _Apache-2.0: https://www.apache.org/licenses/LICENSE-2.0

.. </legal notes>

methods and properties
======================

*)


FUNCTION_BLOCK LTimeAssertionsTests EXTENDS AbstractAssertorTest
VAR
	
END_VAR
VAR CONSTANT
	(* prefix to unify the test names *)
	TEST_NAME_PREFIX			:STRING := 'assert.times.long.';
	(* max value of a LWORD *)
	{attribute 'hide'}
	MAX_LWORD					:LWORD := 16#FFFF_FFFF_FFFF_FFFF;
	(* min value of a LWORD *)
	{attribute 'hide'}
	MIN_LWORD					:LWORD := 16#0000_0000_0000_0000;
	(* only the msb is set *)
	{attribute 'hide'}
	MSB_ONLY					:LWORD := 16#8000_0000_0000_0000;
	(* only the msb is set *)
	{attribute 'hide'}
	LSB_ONLY					:LWORD := 16#0000_0000_0000_0001;
	(* all bits set except the msb *)
	{attribute 'hide'}
	WITHOUT_MSB 				:LWORD := 16#7FFF_FFFF_FFFF_FFFF;
	(* for every nibble is the msb set only *)
	{attribute 'hide'}
	ALL_NIBBLE_MSB				:LWORD := 16#8888_8888_8888_8888;
	(* for every nibble is the msb unset only *)
	{attribute 'hide'}
	WITHOUT_NIBBLE_MSB			:LWORD := 16#7777_7777_7777_7777;
	(* for every nibble is the lsb set only *)
	{attribute 'hide'}
	ALL_NIBBLE_LSB				:LWORD := 16#1111_1111_1111_1111;
	(* every bit is set except the lsb *)
	{attribute 'hide'}
	LSB_IS_UNSET				:LWORD := 16#FFFF_FFFF_FFFF_FFFE;
	(* max vale of time *)
	LTIME_MAX					:LTIME := TO_LTIME(MAX_LWORD);
	(* min vale of time *)
	LTIME_MIN					:LTIME := TO_LTIME(MIN_LWORD);
	(* only the msb is set *)
	LTIME_MSB_ONLY				:LTIME := TO_LTIME(MSB_ONLY);
	(* all bits set except the msb *)
	LTIME_WITHOUT_MSB 			:LTIME := TO_LTIME(WITHOUT_MSB);
	(* for every nibble is the msb set only *)
	LTIME_ALL_NIBBLE_MSB		:LTIME := TO_LTIME(ALL_NIBBLE_MSB);
	(* for every nibble is the msb unset only *)
	LTIME_WITHOUT_NIBBLE_MSB	:LTIME := TO_LTIME(WITHOUT_NIBBLE_MSB);
	(* for every nibble is the lsb set only *)
	LTIME_ALL_NIBBLE_LSB		:LTIME := TO_LTIME(ALL_NIBBLE_LSB);	
	(* every bit is set except the lsb *)
	LTIME_LSB_IS_UNSET			:LTIME := TO_LTIME(LSB_IS_UNSET);
	(* only the msb is set *)
	LTIME_LSB_ONLY				:LTIME := TO_LTIME(LSB_ONLY);
END_VAR

THIS^.runTimeHasExpired();
THIS^.runTimeHasNotExpired();
THIS^.runValueIsEqualToTests();
THIS^.runValueIsGreaterThanTests();
THIS^.runValueIsInRangeOfTests();
THIS^.runValueIsLessThanTests();
THIS^.runValueIsMaxTests();
THIS^.runValueIsMinTests();
THIS^.runValueIsNotEqualToTests();

(*

short summary
==================
This test method is a helper function to create a unified test name

.. <legal notes>

legal notes
=================
| SPDX-FileCopyrightText: © 2022 ekvip automation GmbH <info@ekvip.de>
| SPDX-License-Identifier: Apache-2.0
| For details check: Apache-2.0_

.. _Apache-2.0: https://www.apache.org/licenses/LICENSE-2.0

.. </legal notes>

parameters
==========

*)

METHOD PROTECTED getTestNameFor :Tc2_System.T_MaxString
VAR_INPUT
	(* name of the method to test, to create a unified test name *)
	nameOfMethodToTest	:Tc2_System.T_MaxString;
END_VAR
getTestNameFor := Tc2_Standard.CONCAT(THIS^.TEST_NAME_PREFIX, nameOfMethodToTest);
END_METHOD

(*

short summary
=================
This method returns the passed time since the timestamp was created
(helper method of CNM_AssertionInterfaces)

.. <legal notes>

legal notes
=================
| SPDX-FileCopyrightText: © 2022 ekvip automation GmbH <info@ekvip.de>
| SPDX-License-Identifier: Apache-2.0
| For details check: Apache-2.0_

.. _Apache-2.0: https://www.apache.org/licenses/LICENSE-2.0

.. </legal notes>

parameters
=================
:return: passed time since ``startTime``

*)

METHOD PROTECTED getTimePassed :LTIME
VAR_INPUT
	(* timestamp start *)
	startTime	:LTIME;
END_VAR
VAR
	(* current time to calculate the passed time *)
	currentTime	:LTIME;
END_VAR
currentTime := LTIME();
IF (currentTime > startTime) THEN
	getTimePassed := (currentTime - startTime);
ELSE
	getTimePassed := ((THIS^.LTIME_MAX - startTime) + currentTime);
END_IF
END_METHOD

(*

short summary
==================
This test method tests ``assert.times.long.timeHasExpired``
method of CNM_AssertionInterfaces library with various inputs

.. <legal notes>

legal notes
=================
| SPDX-FileCopyrightText: © 2022 ekvip automation GmbH <info@ekvip.de>
| SPDX-License-Identifier: Apache-2.0
| For details check: Apache-2.0_

.. _Apache-2.0: https://www.apache.org/licenses/LICENSE-2.0

.. </legal notes>

*)

METHOD runTimeHasExpired
RETURN (NOT TcUnit.TEST_ORDERED(THIS^.getTestNameFor('timeHasExpired')));

THIS^.testTimeHasExpired(
	valueToTest := THIS^.LTIME_MAX,
	expiring := THIS^.LTIME_MAX
);
THIS^.testTimeHasExpired(
	valueToTest := THIS^.LTIME_MIN,
	expiring := THIS^.LTIME_MIN
);
THIS^.testTimeHasExpired(
	valueToTest := THIS^.LTIME_MAX,
	expiring := THIS^.LTIME_MIN
);
THIS^.testTimeHasExpired(
	valueToTest := THIS^.LTIME_MIN,
	expiring := THIS^.LTIME_MAX
);
THIS^.testTimeHasExpired(
	valueToTest := THIS^.LTIME_ALL_NIBBLE_LSB,
	expiring := THIS^.LTIME_ALL_NIBBLE_LSB
);	
THIS^.testTimeHasExpired(
	valueToTest := THIS^.LTIME_ALL_NIBBLE_LSB,
	expiring := THIS^.LTIME_ALL_NIBBLE_MSB
);
THIS^.testTimeHasExpired(
	valueToTest := THIS^.LTIME_ALL_NIBBLE_MSB,
	expiring := THIS^.LTIME_ALL_NIBBLE_LSB
);
THIS^.testTimeHasExpired(
	valueToTest := THIS^.LTIME_LSB_ONLY,
	expiring := THIS^.LTIME_MSB_ONLY
);
THIS^.testTimeHasExpired(
	valueToTest := THIS^.LTIME_MSB_ONLY,
	expiring := THIS^.LTIME_MSB_ONLY
);
THIS^.testTimeHasExpired(
	valueToTest := THIS^.LTIME_MSB_ONLY,
	expiring := THIS^.LTIME_LSB_ONLY
);
THIS^.testTimeHasExpired(
	valueToTest := THIS^.LTIME_LSB_IS_UNSET,
	expiring := THIS^.LTIME_MAX
);
THIS^.testTimeHasExpired(
	valueToTest := THIS^.LTIME_MAX,
	expiring := THIS^.LTIME_LSB_IS_UNSET
);

TcUnit.TEST_FINISHED();
END_METHOD

(*

short summary
==================
This test method tests ``assert.times.long.timeHasNotExpired``
method of CNM_AssertionInterfaces library with various inputs

.. <legal notes>

legal notes
=================
| SPDX-FileCopyrightText: © 2022 ekvip automation GmbH <info@ekvip.de>
| SPDX-License-Identifier: Apache-2.0
| For details check: Apache-2.0_

.. _Apache-2.0: https://www.apache.org/licenses/LICENSE-2.0

.. </legal notes>

*)

METHOD runTimeHasNotExpired
RETURN (NOT TcUnit.TEST_ORDERED(THIS^.getTestNameFor('timeHasNotExpired')));

THIS^.testTimeHasExpired(
	valueToTest := THIS^.LTIME_MAX,
	expiring := THIS^.LTIME_MAX
);
THIS^.testTimeHasExpired(
	valueToTest := THIS^.LTIME_MIN,
	expiring := THIS^.LTIME_MIN
);
THIS^.testTimeHasExpired(
	valueToTest := THIS^.LTIME_MAX,
	expiring := THIS^.LTIME_MIN
);
THIS^.testTimeHasExpired(
	valueToTest := THIS^.LTIME_MIN,
	expiring := THIS^.LTIME_MAX
);
THIS^.testTimeHasExpired(
	valueToTest := THIS^.LTIME_ALL_NIBBLE_LSB,
	expiring := THIS^.LTIME_ALL_NIBBLE_LSB
);	
THIS^.testTimeHasExpired(
	valueToTest := THIS^.LTIME_ALL_NIBBLE_LSB,
	expiring := THIS^.LTIME_ALL_NIBBLE_MSB
);
THIS^.testTimeHasExpired(
	valueToTest := THIS^.LTIME_ALL_NIBBLE_MSB,
	expiring := THIS^.LTIME_ALL_NIBBLE_LSB
);
THIS^.testTimeHasExpired(
	valueToTest := THIS^.LTIME_LSB_ONLY,
	expiring := THIS^.LTIME_MSB_ONLY
);
THIS^.testTimeHasExpired(
	valueToTest := THIS^.LTIME_MSB_ONLY,
	expiring := THIS^.LTIME_MSB_ONLY
);
THIS^.testTimeHasExpired(
	valueToTest := THIS^.LTIME_MSB_ONLY,
	expiring := THIS^.LTIME_LSB_ONLY
);
THIS^.testTimeHasExpired(
	valueToTest := THIS^.LTIME_LSB_IS_UNSET,
	expiring := THIS^.LTIME_MAX
);
THIS^.testTimeHasExpired(
	valueToTest := THIS^.LTIME_MAX,
	expiring := THIS^.LTIME_LSB_IS_UNSET
);

TcUnit.TEST_FINISHED();
END_METHOD

(*

short summary
==================
This test method tests ``assert.times.long.valueIsEqualTo``
method of CNM_AssertionInterfaces library with various inputs

.. <legal notes>

legal notes
=================
| SPDX-FileCopyrightText: © 2022 ekvip automation GmbH <info@ekvip.de>
| SPDX-License-Identifier: Apache-2.0
| For details check: Apache-2.0_

.. _Apache-2.0: https://www.apache.org/licenses/LICENSE-2.0

.. </legal notes>

*)

METHOD runValueIsEqualToTests
RETURN (NOT TcUnit.TEST_ORDERED(THIS^.getTestNameFor('valueIsEqualTo')));

THIS^.testValueIsEqualTo(
	valueToTest := THIS^.LTIME_MAX,
	expected := THIS^.LTIME_MAX
);
THIS^.testValueIsEqualTo(
	valueToTest := THIS^.LTIME_MIN,
	expected := THIS^.LTIME_MIN
);
THIS^.testValueIsEqualTo(
	valueToTest := THIS^.LTIME_MIN,
	expected := THIS^.LTIME_MAX
);
THIS^.testValueIsEqualTo(
	valueToTest := THIS^.LTIME_MAX,
	expected := THIS^.LTIME_MIN
);
THIS^.testValueIsEqualTo(
	valueToTest := THIS^.LTIME_ALL_NIBBLE_LSB,
	expected := THIS^.LTIME_ALL_NIBBLE_LSB
);
THIS^.testValueIsEqualTo(
	valueToTest := THIS^.LTIME_LSB_ONLY,
	expected := THIS^.LTIME_MSB_ONLY
);
THIS^.testValueIsEqualTo(
	valueToTest := THIS^.LTIME_MSB_ONLY,
	expected := THIS^.LTIME_MSB_ONLY
);
THIS^.testValueIsEqualTo(
	valueToTest := THIS^.LTIME_MSB_ONLY,
	expected := THIS^.LTIME_LSB_ONLY
);

TcUnit.TEST_FINISHED();
END_METHOD

(*

short summary
==================
This test method tests ``assert.times.long.valueIsGreaterThan``
method of CNM_AssertionInterfaces library with various inputs

.. <legal notes>

legal notes
=================
| SPDX-FileCopyrightText: © 2022 ekvip automation GmbH <info@ekvip.de>
| SPDX-License-Identifier: Apache-2.0
| For details check: Apache-2.0_

.. _Apache-2.0: https://www.apache.org/licenses/LICENSE-2.0

.. </legal notes>

*)

METHOD runValueIsGreaterThanTests
RETURN (NOT TcUnit.TEST_ORDERED(THIS^.getTestNameFor('valueIsGreaterThan')));

THIS^.testValueIsGreaterThan(
	valueToTest := THIS^.LTIME_MAX,
	lessValue := THIS^.LTIME_MAX
);
THIS^.testValueIsGreaterThan(
	valueToTest := THIS^.LTIME_MIN,
	lessValue := THIS^.LTIME_MIN
);
THIS^.testValueIsGreaterThan(
	valueToTest := THIS^.LTIME_MIN,
	lessValue := THIS^.LTIME_MAX
);
THIS^.testValueIsGreaterThan(
	valueToTest := THIS^.LTIME_MAX,
	lessValue := THIS^.LTIME_MIN
);
THIS^.testValueIsGreaterThan(
	valueToTest := THIS^.LTIME_ALL_NIBBLE_LSB,
	lessValue := THIS^.LTIME_ALL_NIBBLE_LSB
);
THIS^.testValueIsGreaterThan(
	valueToTest := THIS^.LTIME_ALL_NIBBLE_MSB,
	lessValue := THIS^.LTIME_ALL_NIBBLE_LSB
);
THIS^.testValueIsGreaterThan(
	valueToTest := THIS^.LTIME_ALL_NIBBLE_LSB,
	lessValue := THIS^.LTIME_ALL_NIBBLE_MSB
);
THIS^.testValueIsGreaterThan(
	valueToTest := THIS^.LTIME_LSB_ONLY,
	lessValue := THIS^.LTIME_MSB_ONLY
);
THIS^.testValueIsGreaterThan(
	valueToTest := THIS^.LTIME_MSB_ONLY,
	lessValue := THIS^.LTIME_MSB_ONLY
);
THIS^.testValueIsGreaterThan(
	valueToTest := THIS^.LTIME_MSB_ONLY,
	lessValue := THIS^.LTIME_LSB_ONLY
);
THIS^.testValueIsGreaterThan(
	valueToTest := THIS^.LTIME_LSB_IS_UNSET,
	lessValue := THIS^.LTIME_MAX
);
THIS^.testValueIsGreaterThan(
	valueToTest := THIS^.LTIME_MAX,
	lessValue := THIS^.LTIME_LSB_IS_UNSET
);

TcUnit.TEST_FINISHED();
END_METHOD

(*

short summary
==================
This test method tests ``assert.times.long.valueIsInRangeOf``
method of CNM_AssertionInterfaces library with various inputs

.. <legal notes>

legal notes
=================
| SPDX-FileCopyrightText: © 2022 ekvip automation GmbH <info@ekvip.de>
| SPDX-License-Identifier: Apache-2.0
| For details check: Apache-2.0_

.. _Apache-2.0: https://www.apache.org/licenses/LICENSE-2.0

.. </legal notes>

*)

METHOD runValueIsInRangeOfTests
RETURN (NOT TcUnit.TEST_ORDERED(THIS^.getTestNameFor('valueIsInRangeOf')));

THIS^.testValueIsInRangeOf(
	lowerLimit := THIS^.LTIME_MIN,
	valueToTest := THIS^.LTIME_MAX,
	upperLimit	:= THIS^.LTIME_MAX
);
THIS^.testValueIsInRangeOf(
	lowerLimit := THIS^.LTIME_MIN,
	valueToTest := THIS^.LTIME_MIN,
	upperLimit	:= THIS^.LTIME_MAX
);
THIS^.testValueIsInRangeOf(
	lowerLimit := THIS^.LTIME_MAX,
	valueToTest := THIS^.LTIME_MAX,
	upperLimit	:= THIS^.LTIME_MIN
);
THIS^.testValueIsInRangeOf(
	lowerLimit := THIS^.LTIME_MAX,
	valueToTest := THIS^.LTIME_MIN,
	upperLimit	:= THIS^.LTIME_MIN
);
THIS^.testValueIsInRangeOf(
	lowerLimit := THIS^.LTIME_LSB_IS_UNSET,
	valueToTest := THIS^.LTIME_MIN,
	upperLimit	:= THIS^.LTIME_MAX
);
THIS^.testValueIsInRangeOf(
	lowerLimit := THIS^.LTIME_MIN,
	valueToTest := THIS^.LTIME_LSB_IS_UNSET,
	upperLimit	:= THIS^.LTIME_MAX
);
THIS^.testValueIsInRangeOf(
	lowerLimit := THIS^.LTIME_LSB_IS_UNSET,
	valueToTest := THIS^.LTIME_LSB_IS_UNSET,
	upperLimit	:= THIS^.LTIME_LSB_IS_UNSET
);
THIS^.testValueIsInRangeOf(
	lowerLimit := THIS^.LTIME_ALL_NIBBLE_LSB,
	valueToTest := THIS^.LTIME_LSB_IS_UNSET,
	upperLimit	:= THIS^.LTIME_ALL_NIBBLE_MSB
);
THIS^.testValueIsInRangeOf(
	lowerLimit := THIS^.LTIME_LSB_IS_UNSET,
	valueToTest := THIS^.LTIME_ALL_NIBBLE_LSB,
	upperLimit	:= THIS^.LTIME_ALL_NIBBLE_MSB
);
THIS^.testValueIsInRangeOf(
	lowerLimit := THIS^.LTIME_LSB_ONLY,
	valueToTest := THIS^.LTIME_WITHOUT_MSB,
	upperLimit	:= THIS^.LTIME_MSB_ONLY
);
THIS^.testValueIsInRangeOf(
	lowerLimit := THIS^.LTIME_WITHOUT_MSB,
	valueToTest := THIS^.LTIME_LSB_ONLY,
	upperLimit	:= THIS^.LTIME_MSB_ONLY
);
THIS^.testValueIsInRangeOf(
	lowerLimit := THIS^.LTIME_WITHOUT_NIBBLE_MSB,
	valueToTest := THIS^.LTIME_MAX,
	upperLimit	:= THIS^.LTIME_ALL_NIBBLE_MSB
);
THIS^.testValueIsInRangeOf(
	lowerLimit := THIS^.LTIME_WITHOUT_NIBBLE_MSB,
	valueToTest := THIS^.LTIME_MIN,
	upperLimit	:= THIS^.LTIME_ALL_NIBBLE_MSB
);
THIS^.testValueIsInRangeOf(
	lowerLimit := THIS^.LTIME_WITHOUT_NIBBLE_MSB,
	valueToTest := THIS^.LTIME_WITHOUT_NIBBLE_MSB,
	upperLimit	:= THIS^.LTIME_ALL_NIBBLE_MSB
);
THIS^.testValueIsInRangeOf(
	lowerLimit := THIS^.LTIME_WITHOUT_NIBBLE_MSB,
	valueToTest := THIS^.LTIME_ALL_NIBBLE_MSB,
	upperLimit	:= THIS^.LTIME_ALL_NIBBLE_MSB
);

TcUnit.TEST_FINISHED();
END_METHOD

(*

short summary
==================
This test method tests ``assert.times.long.valueIsLessThan``
method of CNM_AssertionInterfaces library with various inputs

.. <legal notes>

legal notes
=================
| SPDX-FileCopyrightText: © 2022 ekvip automation GmbH <info@ekvip.de>
| SPDX-License-Identifier: Apache-2.0
| For details check: Apache-2.0_

.. _Apache-2.0: https://www.apache.org/licenses/LICENSE-2.0

.. </legal notes>

*)

METHOD runValueIsLessThanTests
RETURN (NOT TcUnit.TEST_ORDERED(THIS^.getTestNameFor('valueIsLessThan')));

THIS^.testValueIsLessThan(
	valueToTest := THIS^.LTIME_MAX,
	greaterValue := THIS^.LTIME_MAX
);
THIS^.testValueIsLessThan(
	valueToTest := THIS^.LTIME_MIN,
	greaterValue := THIS^.LTIME_MIN
);
THIS^.testValueIsLessThan(
	valueToTest := THIS^.LTIME_MIN,
	greaterValue := THIS^.LTIME_MAX
);
THIS^.testValueIsLessThan(
	valueToTest := THIS^.LTIME_MAX,
	greaterValue := THIS^.LTIME_MIN
);
THIS^.testValueIsLessThan(
	valueToTest := THIS^.LTIME_ALL_NIBBLE_LSB,
	greaterValue := THIS^.LTIME_ALL_NIBBLE_LSB
);
THIS^.testValueIsLessThan(
	valueToTest := THIS^.LTIME_ALL_NIBBLE_MSB,
	greaterValue := THIS^.LTIME_ALL_NIBBLE_LSB
);
THIS^.testValueIsLessThan(
	valueToTest := THIS^.LTIME_ALL_NIBBLE_LSB,
	greaterValue := THIS^.LTIME_ALL_NIBBLE_MSB
);
THIS^.testValueIsLessThan(
	valueToTest := THIS^.LTIME_LSB_ONLY,
	greaterValue := THIS^.LTIME_MSB_ONLY
);
THIS^.testValueIsLessThan(
	valueToTest := THIS^.LTIME_MSB_ONLY,
	greaterValue := THIS^.LTIME_MSB_ONLY
);
THIS^.testValueIsLessThan(
	valueToTest := THIS^.LTIME_MSB_ONLY,
	greaterValue := THIS^.LTIME_LSB_ONLY
);
THIS^.testValueIsLessThan(
	valueToTest := THIS^.LTIME_LSB_IS_UNSET,
	greaterValue := THIS^.LTIME_MAX
);
THIS^.testValueIsLessThan(
	valueToTest := THIS^.LTIME_MAX,
	greaterValue := THIS^.LTIME_LSB_IS_UNSET
);

TcUnit.TEST_FINISHED();
END_METHOD

(*

short summary
==================
This test method tests ``assert.times.long.valueIsMax``
method of CNM_AssertionInterfaces library with various inputs

.. <legal notes>

legal notes
=================
| SPDX-FileCopyrightText: © 2022 ekvip automation GmbH <info@ekvip.de>
| SPDX-License-Identifier: Apache-2.0
| For details check: Apache-2.0_

.. _Apache-2.0: https://www.apache.org/licenses/LICENSE-2.0

.. </legal notes>

*)

METHOD runValueIsMaxTests
RETURN (NOT TcUnit.TEST_ORDERED(THIS^.getTestNameFor('valueIsMax')));

THIS^.testValueIsMax(
	valueToTest := THIS^.LTIME_MAX,
	maximumValue := THIS^.LTIME_MAX
);
THIS^.testValueIsMax(
	valueToTest := THIS^.LTIME_MIN,
	maximumValue := THIS^.LTIME_MIN
);
THIS^.testValueIsMax(
	valueToTest := THIS^.LTIME_MIN,
	maximumValue := THIS^.LTIME_MAX
);
THIS^.testValueIsMax(
	valueToTest := THIS^.LTIME_MAX,
	maximumValue := THIS^.LTIME_MIN
);
THIS^.testValueIsMax(
	valueToTest := THIS^.LTIME_ALL_NIBBLE_LSB,
	maximumValue := THIS^.LTIME_ALL_NIBBLE_LSB
);
THIS^.testValueIsMax(
	valueToTest := THIS^.LTIME_ALL_NIBBLE_MSB,
	maximumValue := THIS^.LTIME_ALL_NIBBLE_LSB
);
THIS^.testValueIsMax(
	valueToTest := THIS^.LTIME_ALL_NIBBLE_LSB,
	maximumValue := THIS^.LTIME_ALL_NIBBLE_MSB
);
THIS^.testValueIsMax(
	valueToTest := THIS^.LTIME_LSB_ONLY,
	maximumValue := THIS^.LTIME_MSB_ONLY
);
THIS^.testValueIsMax(
	valueToTest := THIS^.LTIME_MSB_ONLY,
	maximumValue := THIS^.LTIME_MSB_ONLY
);
THIS^.testValueIsMax(
	valueToTest := THIS^.LTIME_MSB_ONLY,
	maximumValue := THIS^.LTIME_LSB_ONLY
);
THIS^.testValueIsMax(
	valueToTest := THIS^.LTIME_LSB_IS_UNSET,
	maximumValue := THIS^.LTIME_MAX
);
THIS^.testValueIsMax(
	valueToTest := THIS^.LTIME_MAX,
	maximumValue := THIS^.LTIME_LSB_IS_UNSET
);

TcUnit.TEST_FINISHED();
END_METHOD

(*

short summary
==================
This test method tests ``assert.times.long.valueIsMin``
method of CNM_AssertionInterfaces library with various inputs

.. <legal notes>

legal notes
=================
| SPDX-FileCopyrightText: © 2022 ekvip automation GmbH <info@ekvip.de>
| SPDX-License-Identifier: Apache-2.0
| For details check: Apache-2.0_

.. _Apache-2.0: https://www.apache.org/licenses/LICENSE-2.0

.. </legal notes>

*)

METHOD runValueIsMinTests
RETURN (NOT TcUnit.TEST_ORDERED(THIS^.getTestNameFor('valueIsMin')));

THIS^.testValueIsMin(
	valueToTest := THIS^.LTIME_MAX,
	minimumValue := THIS^.LTIME_MAX
);
THIS^.testValueIsMin(
	valueToTest := THIS^.LTIME_MIN,
	minimumValue := THIS^.LTIME_MIN
);
THIS^.testValueIsMin(
	valueToTest := THIS^.LTIME_MIN,
	minimumValue := THIS^.LTIME_MAX
);
THIS^.testValueIsMin(
	valueToTest := THIS^.LTIME_MAX,
	minimumValue := THIS^.LTIME_MIN
);
THIS^.testValueIsMin(
	valueToTest := THIS^.LTIME_ALL_NIBBLE_LSB,
	minimumValue := THIS^.LTIME_ALL_NIBBLE_LSB
);
THIS^.testValueIsMin(
	valueToTest := THIS^.LTIME_ALL_NIBBLE_MSB,
	minimumValue := THIS^.LTIME_ALL_NIBBLE_LSB
);
THIS^.testValueIsMin(
	valueToTest := THIS^.LTIME_ALL_NIBBLE_LSB,
	minimumValue := THIS^.LTIME_ALL_NIBBLE_MSB
);
THIS^.testValueIsMin(
	valueToTest := THIS^.LTIME_LSB_ONLY,
	minimumValue := THIS^.LTIME_MSB_ONLY
);
THIS^.testValueIsMin(
	valueToTest := THIS^.LTIME_MSB_ONLY,
	minimumValue := THIS^.LTIME_MSB_ONLY
);
THIS^.testValueIsMin(
	valueToTest := THIS^.LTIME_MSB_ONLY,
	minimumValue := THIS^.LTIME_LSB_ONLY
);
THIS^.testValueIsMin(
	valueToTest := THIS^.LTIME_LSB_IS_UNSET,
	minimumValue := THIS^.LTIME_MAX
);
THIS^.testValueIsMin(
	valueToTest := THIS^.LTIME_MAX,
	minimumValue := THIS^.LTIME_LSB_IS_UNSET
);
TcUnit.TEST_FINISHED();
END_METHOD

(*

short summary
==================
This test method tests ``assert.times.long.valueIsNotEqualTo``
method of CNM_AssertionInterfaces library with various inputs

.. <legal notes>

legal notes
=================
| SPDX-FileCopyrightText: © 2022 ekvip automation GmbH <info@ekvip.de>
| SPDX-License-Identifier: Apache-2.0
| For details check: Apache-2.0_

.. _Apache-2.0: https://www.apache.org/licenses/LICENSE-2.0

.. </legal notes>

*)

METHOD runValueIsNotEqualToTests
RETURN (NOT TcUnit.TEST_ORDERED(THIS^.getTestNameFor('valueIsNotEqualTo')));

THIS^.testValueIsNotEqualTo(
	valueToTest := THIS^.LTIME_MAX,
	unexpectedValue := THIS^.LTIME_MAX
);
THIS^.testValueIsNotEqualTo(
	valueToTest := THIS^.LTIME_MIN,
	unexpectedValue := THIS^.LTIME_MIN
);
THIS^.testValueIsNotEqualTo(
	valueToTest := THIS^.LTIME_MIN,
	unexpectedValue := THIS^.LTIME_MAX
);
THIS^.testValueIsNotEqualTo(
	valueToTest := THIS^.LTIME_MAX,
	unexpectedValue := THIS^.LTIME_MIN
);
THIS^.testValueIsNotEqualTo(
	valueToTest := THIS^.LTIME_ALL_NIBBLE_LSB,
	unexpectedValue := THIS^.LTIME_ALL_NIBBLE_LSB
);
THIS^.testValueIsNotEqualTo(
	valueToTest := THIS^.LTIME_LSB_ONLY,
	unexpectedValue := THIS^.LTIME_MSB_ONLY
);
THIS^.testValueIsNotEqualTo(
	valueToTest := THIS^.LTIME_MSB_ONLY,
	unexpectedValue := THIS^.LTIME_MSB_ONLY
);
THIS^.testValueIsNotEqualTo(
	valueToTest := THIS^.LTIME_MSB_ONLY,
	unexpectedValue := THIS^.LTIME_LSB_ONLY
);

TcUnit.TEST_FINISHED();
END_METHOD

(*

short summary
==================
This test method tests ``assert.times.long.timeHasExpired``
method of CNM_AssertionInterfaces library, 
it provides the possibility to handover test data via parameter 


.. <legal notes>

legal notes
=================
| SPDX-FileCopyrightText: © 2022 ekvip automation GmbH <info@ekvip.de>
| SPDX-License-Identifier: Apache-2.0
| For details check: Apache-2.0_

.. _Apache-2.0: https://www.apache.org/licenses/LICENSE-2.0

.. </legal notes>

parameters
==========

*)


METHOD testTimeHasExpired 
VAR_INPUT
	(* for the test it's the parameter ``timestamp`` *)
	valueToTest	:LTIME;
	(* for the test it's the parameter ``expiringTime`` *)
	expiring	:LTIME;
END_VAR
VAR
	(* just the expectation if the assertion to test must be wrong or true *)
	assertionIsWrong		:BOOL;
	(* contains the format string for the test message *)
	message					:Tc2_System.T_MaxString;
	(* TwinCAT printf with the test message *)
	messageStringBuilder	:Tc2_Utilities.FB_FormatString;
	(* LTIME value of ``expiringTime`` as string *)
	expiringTimeAsString	:STRING(22);
	(* LTIME value of ``expectedValue`` as string *)
	timestampAsString		:STRING(22);
END_VAR
THIS^.assertorContainer.resetAssertor();

assertionIsWrong := (getTimePassed(startTime := valueToTest) < expiring);

message := SEL(
	assertionIsWrong,
	'timestamp is %s expiringTime is %s assertion must be TRUE', 
	'timestamp is %s expiringTime is %s assertion must be FALSE'
);
timestampAsString := TO_STRING(valueToTest);
expiringTimeAsString := TO_STRING(expiring);

messageStringBuilder(
	sFormat := message,
	arg1 := THIS^.AnyToArg(timestampAsString),
	arg2 := THIS^.AnyToArg(expiringTimeAsString)
);

THIS^.assertorContainer.assertor.assert.times.long.timeHasExpired(
	timestamp		:= valueToTest,
	expiringTime	:= expiring,
	message			:= ''
);

THIS^.AssertEquals_BOOL(
	Expected 	:= assertionIsWrong,
	Actual 		:= THIS^.assertorContainer.wasAssertionWrong,
	Message 	:= messageStringBuilder.sOut
);
END_METHOD

(*

short summary
==================
This test method tests ``assert.times.long.timeHasNotExpired``
method of CNM_AssertionInterfaces library, 
it provides the possibility to handover test data via parameter 


.. <legal notes>

legal notes
=================
| SPDX-FileCopyrightText: © 2022 ekvip automation GmbH <info@ekvip.de>
| SPDX-License-Identifier: Apache-2.0
| For details check: Apache-2.0_

.. _Apache-2.0: https://www.apache.org/licenses/LICENSE-2.0

.. </legal notes>

parameters
==========

*)


METHOD testTimeHasNotExpired 
VAR_INPUT
	(* for the test it's the parameter ``timestamp`` *)
	valueToTest	:LTIME;
	(* for the test it's the parameter ``expiringTime`` *)
	expiring	:LTIME;
END_VAR
VAR
	(* just the expectation if the assertion to test must be wrong or true *)
	assertionIsWrong		:BOOL;
	(* contains the format string for the test message *)
	message					:Tc2_System.T_MaxString;
	(* TwinCAT printf with the test message *)
	messageStringBuilder	:Tc2_Utilities.FB_FormatString;
	(* LTIME value of ``expiringTime`` as string *)
	expiringTimeAsString	:STRING(22);
	(* LTIME value of ``expectedValue`` as string *)
	timestampAsString		:STRING(22);
END_VAR
THIS^.assertorContainer.resetAssertor();

assertionIsWrong := (getTimePassed(startTime := valueToTest) > expiring);

message := SEL(
	assertionIsWrong,
	'timestamp is %s expiringTime is %s assertion must be TRUE', 
	'timestamp is %s expiringTime is %s assertion must be FALSE'
);
timestampAsString := TO_STRING(valueToTest);
expiringTimeAsString := TO_STRING(expiring);

messageStringBuilder(
	sFormat := message,
	arg1 := THIS^.AnyToArg(timestampAsString),
	arg2 := THIS^.AnyToArg(expiringTimeAsString)
);

THIS^.assertorContainer.assertor.assert.times.long.timeHasNotExpired(
	timestamp		:= valueToTest,
	expiringTime	:= expiring,
	message			:= ''
);

